KUKA KRL program: EPS_2_25694_LG04A_A_20260223033044.src

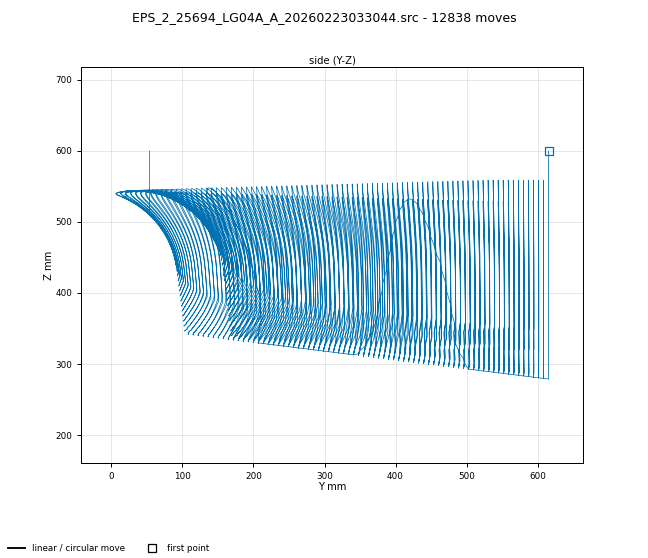
[picture p0: tool path of EPS_2_25694_LG04A_A_20260223033044.src, 12838 of 12840 moves have a stored position in this frame; points joined in program order, loops and branches not executed]
&ACCESS RVP
&REL 4
&COMMENT QRS 19112012
&PARAM EDITMASK = *
DEF PART()
EXT BAS (BAS_COMMAND :IN,REAL :IN )
INT I
BAS (#INITMOV,0 )

;KUKA QRS Post kuka4.cps  Date:22-06-2017 !

File_ID=3043

QRS_PRE_INIT()

;Init var - Until changes are made in qrs_pre_init
Outlet_Square_prg=0
Inlet_1_Square_prg=0
Inlet_2_Square_prg=0
Inlet_3_Square_prg=0
Inlet_4_Square_prg=0
Inlet_5_Square_prg=0

Outlet_1={X 0.000, Y 535.490, Z 458.500, B 0.000, E1 0.000 }
Inlet_1={X 0.000, Y 537.630, Z 428.500, B 0.000, E1 169.000 }
Outlet_1_type=201
Inlet_1_type=201
;QRS#1=Sidecore dimensions
;QRS#2=200-8" PVC SDR 35
;QRS#3=200-8" PVC SDR 35
;QRS#4=
;QRS#5=
;QRS#6=
;QRS#7=
;QRS#8=
;QRS#9=12-08 PSX
;QRS#10=12-08 PSX
;QRS#11=
;QRS#12=
;QRS#13=
;QRS#14=
;QRS#15=
;QRS#16=1220x127x838 2,75'
;QRS#17=EPS Height
;QRS#18=559
;QRS#19=*
;QRS#20= UPDATED VERSION 22-06-2017
;QRS#21=*
Outlet_Square=0100
Inlet_1_Square=0100
Inlet_2_Square=0
Inlet_3_Square=0
Inlet_4_Square=0
Inlet_5_Square=0
Mill_Square=1
Outlet_Square_Prg=204
Inlet_1_Square_prg=204

QRS_INIT()

$ADVANCE=5

; T1
PTP {E1 173.619,E2 173.619}
PTP {X 0,Y 615.493,A -85,B 0,C 180,E1 173.619,E2 173.619,E3 0,E4 0,E5 0,E6 0}
QRS_SPEED_INIT()
LIN {X 0,Y 615.493,Z 600,A -85,B 0,C 180,E1 173.619,E2 173.619,E3 0,E4 0,E5 0,E6 0} C_VEL
LIN {X 0,Y 615.493,Z 288.877,A -85,B 0,C 180,E1 173.619,E2 173.619} C_VEL
LIN {X 0,Y 615.493,Z 280.697,A -85,B 0,C 180,E1 173.619,E2 173.619} C_VEL
LIN {X 0,Y 615.473,Z 278.697,A -85,B 0,C 180,E1 173.433,E2 173.433} C_VEL
LIN {X 0,Y 615.45,Z 278.69,A -85,B 0,C 180,E1 170.8,E2 170.8} C_VEL
LIN {X 0,Y 615.482,Z 278.684,A -85,B 0,C 180,E1 168.139,E2 168.139} C_VEL
LIN {X 0,Y 615.489,Z 278.699,A -85,B 0,C 180,E1 165.451,E2 165.451} C_VEL
LIN {X 0,Y 615.451,Z 278.694,A -85,B 0,C 180,E1 162.728,E2 162.728} C_VEL
LIN {X 0,Y 615.453,Z 278.693,A -85,B 0,C 180,E1 160.661,E2 160.661} C_VEL
LIN {X 0,Y 615.452,Z 278.693,A -85,B 0,C 180,E1 158.567,E2 158.567} C_VEL
LIN {X 0,Y 615.457,Z 278.687,A -85,B 0,C 180,E1 155.998,E2 155.998} C_VEL
LIN {X 0,Y 615.483,Z 278.684,A -85,B 0,C 180,E1 153.555,E2 153.555} C_VEL
LIN {X 0,Y 615.473,Z 278.698,A -85,B 0,C 180,E1 150.593,E2 150.593} C_VEL
LIN {X 0,Y 615.456,Z 278.696,A -85,B 0,C 180,E1 148.312,E2 148.312} C_VEL
LIN {X 0,Y 615.447,Z 278.692,A -85,B 0,C 180,E1 145.975,E2 145.975} C_VEL
LIN {X 0,Y 615.453,Z 278.688,A -85,B 0,C 180,E1 143.572,E2 143.572} C_VEL
LIN {X 0,Y 615.494,Z 278.684,A -85,B 0,C 180,E1 140.937,E2 140.937} C_VEL
LIN {X 0,Y 615.49,Z 278.695,A -85,B 0,C 180,E1 138.526,E2 138.526} C_VEL
LIN {X 0,Y 615.459,Z 278.695,A -85,B 0,C 180,E1 135.847,E2 135.847} C_VEL
LIN {X 0,Y 615.448,Z 278.689,A -85,B 0,C 180,E1 133.248,E2 133.248} C_VEL
LIN {X 0,Y 615.488,Z 278.684,A -85,B 0,C 180,E1 130.607,E2 130.607} C_VEL
LIN {X 0,Y 615.485,Z 278.7,A -85,B 0,C 180,E1 128.011,E2 128.011} C_VEL
LIN {X 0,Y 615.472,Z 278.697,A -85,B 0,C 180,E1 125.617,E2 125.617} C_VEL
LIN {X 0,Y 615.451,Z 278.694,A -85,B 0,C 180,E1 123.239,E2 123.239} C_VEL
LIN {X 0,Y 615.458,Z 278.687,A -85,B 0,C 180,E1 120.541,E2 120.541} C_VEL
LIN {X 0,Y 615.492,Z 278.741,A -85,B 0,C 180,E1 120.207,E2 120.207} C_VEL
LIN {X 0,Y 615.495,Z 297.187,A -85,B 0,C 180,E1 117.177,E2 117.177} C_VEL
LIN {X 0,Y 615.475,Z 314.006,A -85,B 0,C 180,E1 114.452,E2 114.452} C_VEL
LIN {X 0,Y 615.494,Z 318.036,A -85,B 0,C 180,E1 113.809,E2 113.809} C_VEL
LIN {X 0,Y 615.476,Z 425.627,A -85,B 0,C 180,E1 112.53,E2 112.53} C_VEL
LIN {X 0,Y 615.474,Z 438.589,A -85,B 0,C 180,E1 112.239,E2 112.239} C_VEL
LIN {X 0,Y 615.497,Z 450.996,A -85,B 0,C 180,E1 111.828,E2 111.828} C_VEL
LIN {X 0,Y 615.482,Z 463.588,A -85,B 0,C 180,E1 111.257,E2 111.257} C_VEL
LIN {X 0,Y 615.496,Z 475.428,A -85,B 0,C 180,E1 110.558,E2 110.558} C_VEL
LIN {X 0,Y 615.498,Z 483.736,A -85,B 0,C 180,E1 109.946,E2 109.946} C_VEL
LIN {X 0,Y 615.498,Z 490.882,A -85,B 0,C 180,E1 109.338,E2 109.338} C_VEL
LIN {X 0,Y 615.496,Z 499.643,A -85,B 0,C 180,E1 108.444,E2 108.444} C_VEL
LIN {X 0,Y 615.493,Z 507.562,A -85,B 0,C 180,E1 107.442,E2 107.442} C_VEL
LIN {X 0,Y 615.496,Z 513.912,A -85,B 0,C 180,E1 106.432,E2 106.432} C_VEL
LIN {X 0,Y 615.497,Z 519.787,A -85,B 0,C 180,E1 105.226,E2 105.226} C_VEL
LIN {X 0,Y 615.496,Z 522.37,A -85,B 0,C 180,E1 104.549,E2 104.549} C_VEL
LIN {X 0,Y 615.496,Z 524.427,A -85,B 0,C 180,E1 103.874,E2 103.874} C_VEL
LIN {X 0,Y 615.495,Z 526.05,A -85,B 0,C 180,E1 103.201,E2 103.201} C_VEL
LIN {X 0,Y 615.497,Z 527.253,A -85,B 0,C 180,E1 102.53,E2 102.53} C_VEL
LIN {X 0,Y 615.494,Z 527.997,A -85,B 0,C 180,E1 101.861,E2 101.861} C_VEL
LIN {X 0,Y 615.497,Z 528.293,A -85,B 0,C 180,E1 100.527,E2 100.527} C_VEL
LIN {X 0,Y 615.496,Z 527.836,A -85,B 0,C 180,E1 99.862,E2 99.862} C_VEL
LIN {X 0,Y 615.495,Z 525.678,A -85,B 0,C 180,E1 98.537,E2 98.537} C_VEL
LIN {X 0,Y 615.495,Z 522.962,A -85,B 0,C 180,E1 97.546,E2 97.546} C_VEL
LIN {X 0,Y 615.497,Z 519.242,A -85,B 0,C 180,E1 96.557,E2 96.557} C_VEL
LIN {X 0,Y 615.497,Z 514.417,A -85,B 0,C 180,E1 95.57,E2 95.57} C_VEL
LIN {X 0,Y 615.495,Z 508.351,A -85,B 0,C 180,E1 94.585,E2 94.585} C_VEL
LIN {X 0,Y 615.493,Z 500.832,A -85,B 0,C 180,E1 93.601,E2 93.601} C_VEL
LIN {X 0,Y 615.498,Z 493.027,A -85,B 0,C 180,E1 92.782,E2 92.782} C_VEL
LIN {X 0,Y 615.497,Z 485.721,A -85,B 0,C 180,E1 92.127,E2 92.127} C_VEL
LIN {X 0,Y 615.486,Z 477.224,A -85,B 0,C 180,E1 91.473,E2 91.473} C_VEL
LIN {X 0,Y 615.483,Z 466.689,A -85,B 0,C 180,E1 90.818,E2 90.818} C_VEL
LIN {X 0,Y 615.492,Z 454.96,A -85,B 0,C 180,E1 90.246,E2 90.246} C_VEL
LIN {X 0,Y 615.484,Z 442.825,A -85,B 0,C 180,E1 89.796,E2 89.796} C_VEL
LIN {X 0,Y 615.474,Z 430.38,A -85,B 0,C 180,E1 89.469,E2 89.469} C_VEL
LIN {X 0,Y 615.478,Z 415.696,A -85,B 0,C 180,E1 89.244,E2 89.244} C_VEL
LIN {X 0,Y 615.496,Z 317.979,A -85,B 0,C 180,E1 88.099,E2 88.099} C_VEL
LIN {X 0,Y 615.475,Z 300.382,A -85,B 0,C 180,E1 85.252,E2 85.252} C_VEL
LIN {X 0,Y 615.496,Z 283.292,A -85,B 0,C 180,E1 82.455,E2 82.455} C_VEL
LIN {X 0,Y 615.44,Z 278.695,A -85,B 0,C 180,E1 81.67,E2 81.67} C_VEL
LIN {X 0,Y 615.441,Z 278.691,A -85,B 0,C 180,E1 79.137,E2 79.137} C_VEL
LIN {X 0,Y 615.457,Z 278.69,A -85,B 0,C 180,E1 76.799,E2 76.799} C_VEL
LIN {X 0,Y 615.491,Z 278.699,A -85,B 0,C 180,E1 74.096,E2 74.096} C_VEL
LIN {X 0,Y 615.436,Z 278.696,A -85,B 0,C 180,E1 71.353,E2 71.353} C_VEL
LIN {X 0,Y 615.435,Z 278.696,A -85,B 0,C 180,E1 69.268,E2 69.268} C_VEL
LIN {X 0,Y 615.432,Z 278.696,A -85,B 0,C 180,E1 67.154,E2 67.154} C_VEL
LIN {X 0,Y 615.428,Z 278.695,A -85,B 0,C 180,E1 65.006,E2 65.006} C_VEL
LIN {X 0,Y 615.425,Z 278.695,A -85,B 0,C 180,E1 62.821,E2 62.821} C_VEL
LIN {X 0,Y 615.426,Z 278.694,A -85,B 0,C 180,E1 60.591,E2 60.591} C_VEL
LIN {X 0,Y 615.431,Z 278.694,A -85,B 0,C 180,E1 58.312,E2 58.312} C_VEL
LIN {X 0,Y 615.456,Z 278.693,A -85,B 0,C 180,E1 55.977,E2 55.977} C_VEL
LIN {X 0,Y 615.456,Z 278.699,A -85,B 0,C 180,E1 53.068,E2 53.068} C_VEL
LIN {X 0,Y 615.419,Z 278.696,A -85,B 0,C 180,E1 50.246,E2 50.246} C_VEL
LIN {X 0,Y 615.455,Z 278.694,A -85,B 0,C 180,E1 47.645,E2 47.645} C_VEL
LIN {X 0,Y 615.472,Z 278.7,A -85,B 0,C 180,E1 44.931,E2 44.931} C_VEL
LIN {X 0,Y 615.42,Z 278.698,A -85,B 0,C 180,E1 42.359,E2 42.359} C_VEL
LIN {X 0,Y 615.41,Z 278.698,A -85,B 0,C 180,E1 40.082,E2 40.082} C_VEL
LIN {X 0,Y 615.41,Z 278.698,A -85,B 0,C 180,E1 38.004,E2 38.004} C_VEL
LIN {X 0,Y 615.413,Z 278.698,A -85,B 0,C 180,E1 35.621,E2 35.621} C_VEL
LIN {X 0,Y 615.434,Z 278.698,A -85,B 0,C 180,E1 33.24,E2 33.24} C_VEL
LIN {X 0,Y 615.431,Z 278.7,A -85,B 0,C 180,E1 30.164,E2 30.164} C_VEL
LIN {X 0,Y 615.415,Z 278.7,A -85,B 0,C 180,E1 27.919,E2 27.919} C_VEL
LIN {X 0,Y 615.402,Z 278.7,A -85,B 0,C 180,E1 25.554,E2 25.554} C_VEL
LIN {X 0,Y 615.403,Z 278.7,A -85,B 0,C 180,E1 23.56,E2 23.56} C_VEL
LIN {X 0,Y 615.403,Z 278.7,A -85,B 0,C 180,E1 21.435,E2 21.435} C_VEL
LIN {X 0,Y 615.403,Z 278.7,A -85,B 0,C 180,E1 19.341,E2 19.341} C_VEL
LIN {X 0,Y 615.405,Z 278.699,A -85,B 0,C 180,E1 17.273,E2 17.273} C_VEL
LIN {X 0,Y 615.407,Z 278.699,A -85,B 0,C 180,E1 15.228,E2 15.228} C_VEL
LIN {X 0,Y 615.41,Z 278.698,A -85,B 0,C 180,E1 13.203,E2 13.203} C_VEL
LIN {X 0,Y 615.41,Z 278.698,A -85,B 0,C 180,E1 10.856,E2 10.856} C_VEL
LIN {X 0,Y 615.423,Z 278.699,A -85,B 0,C 180,E1 8.538,E2 8.538} C_VEL
LIN {X 0,Y 615.493,Z 278.7,A -85,B 0,C 180,E1 5.899,E2 5.899} C_VEL
LIN {X 0,Y 615.447,Z 278.695,A -85,B 0,C 180,E1 3.273,E2 3.273} C_VEL
LIN {X 0,Y 615.416,Z 278.697,A -85,B 0,C 180,E1 0.654,E2 0.654} C_VEL
LIN {X 0,Y 615.419,Z 278.696,A -85,B 0,C 180,E1 -1.309,E2 -1.309} C_VEL
LIN {X 0,Y 615.425,Z 278.695,A -85,B 0,C 180,E1 -3.273,E2 -3.273} C_VEL
LIN {X 0,Y 615.431,Z 278.695,A -85,B 0,C 180,E1 -5.242,E2 -5.242} C_VEL
LIN {X 0,Y 615.441,Z 278.694,A -85,B 0,C 180,E1 -7.216,E2 -7.216} C_VEL
LIN {X 0,Y 615.452,Z 278.693,A -85,B 0,C 180,E1 -9.199,E2 -9.199} C_VEL
LIN {X 0,Y 615.462,Z 278.692,A -85,B 0,C 180,E1 -11.193,E2 -11.193} C_VEL
LIN {X 0,Y 615.425,Z 278.695,A -85,B 0,C 180,E1 -13.913,E2 -13.913} C_VEL
LIN {X 0,Y 615.444,Z 278.697,A -85,B 0,C 180,E1 -16.421,E2 -16.421} C_VEL
LIN {X 0,Y 615.482,Z 278.69,A -85,B 0,C 180,E1 -19.338,E2 -19.338} C_VEL
LIN {X 0,Y 615.43,Z 278.694,A -85,B 0,C 180,E1 -22.139,E2 -22.139} C_VEL
LIN {X 0,Y 615.43,Z 278.694,A -85,B 0,C 180,E1 -24.274,E2 -24.274} C_VEL
LIN {X 0,Y 615.433,Z 278.694,A -85,B 0,C 180,E1 -26.447,E2 -26.447} C_VEL
LIN {X 0,Y 615.492,Z 278.696,A -85,B 0,C 180,E1 -29.406,E2 -29.406} C_VEL
LIN {X 0,Y 615.441,Z 278.691,A -85,B 0,C 180,E1 -32.326,E2 -32.326} C_VEL
LIN {X 0,Y 615.437,Z 278.693,A -85,B 0,C 180,E1 -34.696,E2 -34.696} C_VEL
LIN {X 0,Y 615.464,Z 278.697,A -85,B 0,C 180,E1 -37.244,E2 -37.244} C_VEL
LIN {X 0,Y 615.495,Z 278.685,A -85,B 0,C 180,E1 -40.091,E2 -40.091} C_VEL
LIN {X 0,Y 615.469,Z 278.687,A -85,B 0,C 180,E1 -42.355,E2 -42.355} C_VEL
LIN {X 0,Y 615.442,Z 278.691,A -85,B 0,C 180,E1 -44.928,E2 -44.928} C_VEL
LIN {X 0,Y 615.443,Z 278.691,A -85,B 0,C 180,E1 -46.957,E2 -46.957} C_VEL
LIN {X 0,Y 615.448,Z 278.695,A -85,B 0,C 180,E1 -49.392,E2 -49.392} C_VEL
LIN {X 0,Y 615.482,Z 278.704,A -85,B 0,C 180,E1 -51.989,E2 -51.989} C_VEL
LIN {X 0,Y 615.493,Z 278.69,A -85,B 0,C 180,E1 -54.386,E2 -54.386} C_VEL
LIN {X 0,Y 615.485,Z 278.684,A -85,B 0,C 180,E1 -56.765,E2 -56.765} C_VEL
LIN {X 0,Y 615.468,Z 278.685,A -85,B 0,C 180,E1 -59.08,E2 -59.08} C_VEL
LIN {X 0,Y 615.451,Z 278.69,A -85,B 0,C 180,E1 -61.556,E2 -61.556} C_VEL
LIN {X 0,Y 615.451,Z 278.689,A -85,B 0,C 180,E1 -63.555,E2 -63.555} C_VEL
LIN {X 0,Y 615.459,Z 278.694,A -85,B 0,C 180,E1 -65.998,E2 -65.998} C_VEL
LIN {X 0,Y 615.454,Z 278.771,A -85,B 0,C 180,E1 -67.838,E2 -67.838} C_VEL
LIN {X 0,Y 615.483,Z 297.824,A -85,B 0,C 180,E1 -70.489,E2 -70.489} C_VEL
LIN {X 0,Y 615.496,Z 319.189,A -85,B 0,C 180,E1 -73.414,E2 -73.414} C_VEL
LIN {X 0,Y 615.486,Z 340.532,A -85,B 0,C 180,E1 -76.295,E2 -76.295} C_VEL
LIN {X 0,Y 615.476,Z 346.647,A -85,B 0,C 180,E1 -77.114,E2 -77.114} C_VEL
LIN {X 0,Y 615.488,Z 454.864,A -85,B 0,C 180,E1 -78.411,E2 -78.411} C_VEL
LIN {X 0,Y 615.493,Z 467.365,A -85,B 0,C 180,E1 -78.683,E2 -78.683} C_VEL
LIN {X 0,Y 615.492,Z 480.561,A -85,B 0,C 180,E1 -79.111,E2 -79.111} C_VEL
LIN {X 0,Y 615.489,Z 492.488,A -85,B 0,C 180,E1 -79.64,E2 -79.64} C_VEL
LIN {X 0,Y 615.478,Z 504.006,A -85,B 0,C 180,E1 -80.304,E2 -80.304} C_VEL
LIN {X 0,Y 615.498,Z 513.228,A -85,B 0,C 180,E1 -80.968,E2 -80.968} C_VEL
LIN {X 0,Y 615.498,Z 521.008,A -85,B 0,C 180,E1 -81.629,E2 -81.629} C_VEL
LIN {X 0,Y 615.497,Z 530.611,A -85,B 0,C 180,E1 -82.62,E2 -82.62} C_VEL
LIN {X 0,Y 615.49,Z 538.208,A -85,B 0,C 180,E1 -83.609,E2 -83.609} C_VEL
LIN {X 0,Y 615.498,Z 545.207,A -85,B 0,C 180,E1 -84.759,E2 -84.759} C_VEL
LIN {X 0,Y 615.493,Z 549.854,A -85,B 0,C 180,E1 -85.744,E2 -85.744} C_VEL
LIN {X 0,Y 615.496,Z 553.4,A -85,B 0,C 180,E1 -86.728,E2 -86.728} C_VEL
LIN {X 0,Y 615.497,Z 555.234,A -85,B 0,C 180,E1 -87.383,E2 -87.383} C_VEL
LIN {X 0,Y 615.496,Z 556.609,A -85,B 0,C 180,E1 -88.037,E2 -88.037} C_VEL
LIN {X 0,Y 615.496,Z 558.174,A -85,B 0,C 180,E1 -89.346,E2 -89.346} C_VEL
LIN {X 0,Y 615.494,Z 558.389,A -85,B 0,C 180,E1 -90,E2 -90} C_VEL
LIN {X 0,Y 615.496,Z 557.579,A -85,B 0,C 180,E1 -91.309,E2 -91.309} C_VEL
LIN {X 0,Y 615.496,Z 556.607,A -85,B 0,C 180,E1 -91.964,E2 -91.964} C_VEL
LIN {X 0,Y 615.497,Z 555.232,A -85,B 0,C 180,E1 -92.618,E2 -92.618} C_VEL
LIN {X 0,Y 615.496,Z 552.348,A -85,B 0,C 180,E1 -93.601,E2 -93.601} C_VEL
LIN {X 0,Y 615.498,Z 548.44,A -85,B 0,C 180,E1 -94.585,E2 -94.585} C_VEL
LIN {X 0,Y 615.499,Z 543.402,A -85,B 0,C 180,E1 -95.57,E2 -95.57} C_VEL
LIN {X 0,Y 615.489,Z 536.916,A -85,B 0,C 180,E1 -96.577,E2 -96.577} C_VEL
LIN {X 0,Y 615.497,Z 529.129,A -85,B 0,C 180,E1 -97.546,E2 -97.546} C_VEL
LIN {X 0,Y 615.498,Z 519.253,A -85,B 0,C 180,E1 -98.537,E2 -98.537} C_VEL
LIN {X 0,Y 615.492,Z 507.705,A -85,B 0,C 180,E1 -99.448,E2 -99.448} C_VEL
LIN {X 0,Y 615.48,Z 497.148,A -85,B 0,C 180,E1 -100.112,E2 -100.112} C_VEL
LIN {X 0,Y 615.496,Z 484.986,A -85,B 0,C 180,E1 -100.708,E2 -100.708} C_VEL
LIN {X 0,Y 615.489,Z 472.933,A -85,B 0,C 180,E1 -101.155,E2 -101.155} C_VEL
LIN {X 0,Y 615.491,Z 460.398,A -85,B 0,C 180,E1 -101.485,E2 -101.485} C_VEL
LIN {X 0,Y 615.487,Z 447.127,A -85,B 0,C 180,E1 -101.694,E2 -101.694} C_VEL
LIN {X 0,Y 615.475,Z 346.64,A -85,B 0,C 180,E1 -102.887,E2 -102.887} C_VEL
LIN {X 0,Y 615.496,Z 325.462,A -85,B 0,C 180,E1 -105.735,E2 -105.735} C_VEL
LIN {X 0,Y 615.486,Z 304.105,A -85,B 0,C 180,E1 -108.646,E2 -108.646} C_VEL
LIN {X 0,Y 615.497,Z 283.978,A -85,B 0,C 180,E1 -111.432,E2 -111.432} C_VEL
LIN {X 0,Y 615.454,Z 278.69,A -85,B 0,C 180,E1 -112.188,E2 -112.188} C_VEL
LIN {X 0,Y 615.492,Z 278.682,A -85,B 0,C 180,E1 -114.992,E2 -114.992} C_VEL
LIN {X 0,Y 615.478,Z 278.697,A -85,B 0,C 180,E1 -117.916,E2 -117.916} C_VEL
LIN {X 0,Y 615.465,Z 278.695,A -85,B 0,C 180,E1 -120.162,E2 -120.162} C_VEL
LIN {X 0,Y 615.455,Z 278.692,A -85,B 0,C 180,E1 -122.46,E2 -122.46} C_VEL
LIN {X 0,Y 615.455,Z 278.688,A -85,B 0,C 180,E1 -124.817,E2 -124.817} C_VEL
LIN {X 0,Y 615.476,Z 278.683,A -85,B 0,C 180,E1 -127.243,E2 -127.243} C_VEL
LIN {X 0,Y 615.495,Z 278.697,A -85,B 0,C 180,E1 -130.09,E2 -130.09} C_VEL
LIN {X 0,Y 615.49,Z 278.699,A -85,B 0,C 180,E1 -132.353,E2 -132.353} C_VEL
LIN {X 0,Y 615.45,Z 278.691,A -85,B 0,C 180,E1 -135.072,E2 -135.072} C_VEL
LIN {X 0,Y 615.497,Z 278.682,A -85,B 0,C 180,E1 -137.919,E2 -137.919} C_VEL
LIN {X 0,Y 615.49,Z 278.69,A -85,B 0,C 180,E1 -140.25,E2 -140.25} C_VEL
LIN {X 0,Y 615.462,Z 278.695,A -85,B 0,C 180,E1 -143.067,E2 -143.067} C_VEL
LIN {X 0,Y 615.454,Z 278.693,A -85,B 0,C 180,E1 -145.304,E2 -145.304} C_VEL
LIN {X 0,Y 615.453,Z 278.689,A -85,B 0,C 180,E1 -147.674,E2 -147.674} C_VEL
LIN {X 0,Y 615.482,Z 278.683,A -85,B 0,C 180,E1 -150.206,E2 -150.206} C_VEL
LIN {X 0,Y 615.492,Z 278.697,A -85,B 0,C 180,E1 -152.954,E2 -152.954} C_VEL
LIN {X 0,Y 615.452,Z 278.692,A -85,B 0,C 180,E1 -155.726,E2 -155.726} C_VEL
LIN {X 0,Y 615.452,Z 278.692,A -85,B 0,C 180,E1 -157.862,E2 -157.862} C_VEL
LIN {X 0,Y 615.45,Z 278.692,A -85,B 0,C 180,E1 -159.966,E2 -159.966} C_VEL
LIN {X 0,Y 615.451,Z 278.691,A -85,B 0,C 180,E1 -162.042,E2 -162.042} C_VEL
LIN {X 0,Y 615.483,Z 278.683,A -85,B 0,C 180,E1 -164.774,E2 -164.774} C_VEL
LIN {X 0,Y 615.489,Z 278.697,A -85,B 0,C 180,E1 -167.47,E2 -167.47} C_VEL
LIN {X 0,Y 615.458,Z 278.694,A -85,B 0,C 180,E1 -170.137,E2 -170.137} C_VEL
LIN {X 0,Y 615.458,Z 278.687,A -85,B 0,C 180,E1 -172.784,E2 -172.784} C_VEL
LIN {X 0,Y 615.495,Z 278.684,A -85,B 0,C 180,E1 -175.416,E2 -175.416} C_VEL
LIN {X 0,Y 615.496,Z 278.7,A -85,B 0,C 180,E1 -178.037,E2 -178.037} C_VEL
LIN {X 0,Y 615.453,Z 278.693,A -85,B 0,C 180,E1 -180.654,E2 -180.654} C_VEL
LIN {X 0,Y 615.462,Z 278.686,A -85,B 0,C 180,E1 -183.273,E2 -183.273} C_VEL
LIN {X 0,Y 615.493,Z 278.687,A -85,B 0,C 180,E1 -185.899,E2 -185.899} C_VEL
LIN {X 0,Y 615.473,Z 278.697,A -85,B 0,C 180,E1 -186.567,E2 -186.567} C_VEL
LIN {X 0,Y 614.78,Z 278.837,A -85,B 0,C 180,E1 -187.113,E2 -187.113} C_VEL
LIN {X 0,Y 611.93,Z 279.257,A -85,B 0,C 180,E1 -187.999,E2 -187.999} C_VEL
LIN {X 0,Y 609.542,Z 279.564,A -85,B 0,C 180,E1 -188.712,E2 -188.712} C_VEL
LIN {X 0,Y 608.522,Z 279.679,A -85,B 0,C 180,E1 -189.261,E2 -189.261} C_VEL
LIN {X 0,Y 608.441,Z 279.687,A -85,B 0,C 180,E1 -189.447,E2 -189.447} C_VEL
LIN {X 0,Y 608.46,Z 279.688,A -85,B 0,C 180,E1 -192,E2 -192} C_VEL
LIN {X 0,Y 608.469,Z 279.695,A -85,B 0,C 180,E1 -194.721,E2 -194.721} C_VEL
LIN {X 0,Y 608.425,Z 279.69,A -85,B 0,C 180,E1 -197.478,E2 -197.478} C_VEL
LIN {X 0,Y 608.428,Z 279.69,A -85,B 0,C 180,E1 -199.572,E2 -199.572} C_VEL
LIN {X 0,Y 608.443,Z 279.688,A -85,B 0,C 180,E1 -201.693,E2 -201.693} C_VEL
LIN {X 0,Y 608.454,Z 279.69,A -85,B 0,C 180,E1 -204.571,E2 -204.571} C_VEL
LIN {X 0,Y 608.435,Z 279.693,A -85,B 0,C 180,E1 -207.519,E2 -207.519} C_VEL
LIN {X 0,Y 608.419,Z 279.691,A -85,B 0,C 180,E1 -209.964,E2 -209.964} C_VEL
LIN {X 0,Y 608.445,Z 279.687,A -85,B 0,C 180,E1 -212.52,E2 -212.52} C_VEL
LIN {X 0,Y 608.442,Z 279.696,A -85,B 0,C 180,E1 -215.278,E2 -215.278} C_VEL
LIN {X 0,Y 608.452,Z 279.694,A -85,B 0,C 180,E1 -217.748,E2 -217.748} C_VEL
LIN {X 0,Y 608.435,Z 279.689,A -85,B 0,C 180,E1 -220.327,E2 -220.327} C_VEL
LIN {X 0,Y 608.483,Z 279.686,A -85,B 0,C 180,E1 -223.31,E2 -223.31} C_VEL
LIN {X 0,Y 608.459,Z 279.692,A -85,B 0,C 180,E1 -226.129,E2 -226.129} C_VEL
LIN {X 0,Y 608.421,Z 279.69,A -85,B 0,C 180,E1 -228.82,E2 -228.82} C_VEL
LIN {X 0,Y 608.465,Z 279.691,A -85,B 0,C 180,E1 -231.761,E2 -231.761} C_VEL
LIN {X 0,Y 608.425,Z 279.692,A -85,B 0,C 180,E1 -234.721,E2 -234.721} C_VEL
LIN {X 0,Y 608.453,Z 279.687,A -85,B 0,C 180,E1 -237.48,E2 -237.48} C_VEL
LIN {X 0,Y 608.492,Z 279.837,A -85,B 0,C 180,E1 -239.737,E2 -239.737} C_VEL
LIN {X 0,Y 608.484,Z 296.397,A -85,B 0,C 180,E1 -242.483,E2 -242.483} C_VEL
LIN {X 0,Y 608.46,Z 313.301,A -85,B 0,C 180,E1 -245.247,E2 -245.247} C_VEL
LIN {X 0,Y 608.462,Z 318.194,A -85,B 0,C 180,E1 -246.041,E2 -246.041} C_VEL
LIN {X 0,Y 608.525,Z 425.131,A -85,B 0,C 180,E1 -247.325,E2 -247.325} C_VEL
LIN {X 0,Y 608.516,Z 438.538,A -85,B 0,C 180,E1 -247.626,E2 -247.626} C_VEL
LIN {X 0,Y 608.534,Z 451.048,A -85,B 0,C 180,E1 -248.043,E2 -248.043} C_VEL
LIN {X 0,Y 608.488,Z 462.858,A -85,B 0,C 180,E1 -248.576,E2 -248.576} C_VEL
LIN {X 0,Y 608.512,Z 473.869,A -85,B 0,C 180,E1 -249.215,E2 -249.215} C_VEL
LIN {X 0,Y 608.477,Z 483.424,A -85,B 0,C 180,E1 -249.902,E2 -249.902} C_VEL
LIN {X 0,Y 608.487,Z 491.598,A -85,B 0,C 180,E1 -250.606,E2 -250.606} C_VEL
LIN {X 0,Y 608.474,Z 500.264,A -85,B 0,C 180,E1 -251.5,E2 -251.5} C_VEL
LIN {X 0,Y 608.448,Z 508.244,A -85,B 0,C 180,E1 -252.523,E2 -252.523} C_VEL
LIN {X 0,Y 608.434,Z 514.264,A -85,B 0,C 180,E1 -253.483,E2 -253.483} C_VEL
LIN {X 0,Y 608.427,Z 519.744,A -85,B 0,C 180,E1 -254.593,E2 -254.593} C_VEL
LIN {X 0,Y 608.428,Z 523.592,A -85,B 0,C 180,E1 -255.62,E2 -255.62} C_VEL
LIN {X 0,Y 608.438,Z 526.355,A -85,B 0,C 180,E1 -256.643,E2 -256.643} C_VEL
LIN {X 0,Y 608.42,Z 527.637,A -85,B 0,C 180,E1 -257.322,E2 -257.322} C_VEL
LIN {X 0,Y 608.44,Z 528.506,A -85,B 0,C 180,E1 -257.999,E2 -257.999} C_VEL
LIN {X 0,Y 608.448,Z 529,A -85,B 0,C 180,E1 -259.057,E2 -259.057} C_VEL
LIN {X 0,Y 608.432,Z 528.562,A -85,B 0,C 180,E1 -260.022,E2 -260.022} C_VEL
LIN {X 0,Y 608.423,Z 527.762,A -85,B 0,C 180,E1 -260.693,E2 -260.693} C_VEL
LIN {X 0,Y 608.421,Z 526.538,A -85,B 0,C 180,E1 -261.363,E2 -261.363} C_VEL
LIN {X 0,Y 608.424,Z 523.924,A -85,B 0,C 180,E1 -262.366,E2 -262.366} C_VEL
LIN {X 0,Y 608.453,Z 519.172,A -85,B 0,C 180,E1 -263.631,E2 -263.631} C_VEL
LIN {X 0,Y 608.462,Z 513.763,A -85,B 0,C 180,E1 -264.698,E2 -264.698} C_VEL
LIN {X 0,Y 608.438,Z 507.355,A -85,B 0,C 180,E1 -265.694,E2 -265.694} C_VEL
LIN {X 0,Y 608.451,Z 499.384,A -85,B 0,C 180,E1 -266.689,E2 -266.689} C_VEL
LIN {X 0,Y 608.484,Z 489.512,A -85,B 0,C 180,E1 -267.683,E2 -267.683} C_VEL
LIN {X 0,Y 608.471,Z 478.058,A -85,B 0,C 180,E1 -268.593,E2 -268.593} C_VEL
LIN {X 0,Y 608.498,Z 467.652,A -85,B 0,C 180,E1 -269.255,E2 -269.255} C_VEL
LIN {X 0,Y 608.509,Z 456.141,A -85,B 0,C 180,E1 -269.834,E2 -269.834} C_VEL
LIN {X 0,Y 608.517,Z 443.034,A -85,B 0,C 180,E1 -270.33,E2 -270.33} C_VEL
LIN {X 0,Y 608.516,Z 430.618,A -85,B 0,C 180,E1 -270.661,E2 -270.661} C_VEL
LIN {X 0,Y 608.53,Z 417.842,A -85,B 0,C 180,E1 -270.868,E2 -270.868} C_VEL
LIN {X 0,Y 608.498,Z 318.287,A -85,B 0,C 180,E1 -272.047,E2 -272.047} C_VEL
LIN {X 0,Y 608.471,Z 301.29,A -85,B 0,C 180,E1 -274.803,E2 -274.803} C_VEL
LIN {X 0,Y 608.514,Z 284.155,A -85,B 0,C 180,E1 -277.632,E2 -277.632} C_VEL
LIN {X 0,Y 608.42,Z 279.693,A -85,B 0,C 180,E1 -278.385,E2 -278.385} C_VEL
LIN {X 0,Y 608.437,Z 279.688,A -85,B 0,C 180,E1 -280.938,E2 -280.938} C_VEL
LIN {X 0,Y 608.48,Z 279.692,A -85,B 0,C 180,E1 -284.019,E2 -284.019} C_VEL
LIN {X 0,Y 608.414,Z 279.692,A -85,B 0,C 180,E1 -286.784,E2 -286.784} C_VEL
LIN {X 0,Y 608.433,Z 279.691,A -85,B 0,C 180,E1 -289.57,E2 -289.57} C_VEL
LIN {X 0,Y 608.431,Z 279.695,A -85,B 0,C 180,E1 -292.469,E2 -292.469} C_VEL
LIN {X 0,Y 608.432,Z 279.694,A -85,B 0,C 180,E1 -294.571,E2 -294.571} C_VEL
LIN {X 0,Y 608.41,Z 279.692,A -85,B 0,C 180,E1 -297.194,E2 -297.194} C_VEL
LIN {X 0,Y 608.449,Z 279.69,A -85,B 0,C 180,E1 -299.968,E2 -299.968} C_VEL
LIN {X 0,Y 608.431,Z 279.694,A -85,B 0,C 180,E1 -302.88,E2 -302.88} C_VEL
LIN {X 0,Y 608.401,Z 279.694,A -85,B 0,C 180,E1 -305.279,E2 -305.279} C_VEL
LIN {X 0,Y 608.402,Z 279.693,A -85,B 0,C 180,E1 -307.75,E2 -307.75} C_VEL
LIN {X 0,Y 608.43,Z 279.693,A -85,B 0,C 180,E1 -310.326,E2 -310.326} C_VEL
LIN {X 0,Y 608.434,Z 279.692,A -85,B 0,C 180,E1 -313.305,E2 -313.305} C_VEL
LIN {X 0,Y 608.396,Z 279.694,A -85,B 0,C 180,E1 -315.741,E2 -315.741} C_VEL
LIN {X 0,Y 608.397,Z 279.693,A -85,B 0,C 180,E1 -317.933,E2 -317.933} C_VEL
LIN {X 0,Y 608.428,Z 279.694,A -85,B 0,C 180,E1 -320.706,E2 -320.706} C_VEL
LIN {X 0,Y 608.445,Z 279.698,A -85,B 0,C 180,E1 -323.084,E2 -323.084} C_VEL
LIN {X 0,Y 608.447,Z 279.693,A -85,B 0,C 180,E1 -325.529,E2 -325.529} C_VEL
LIN {X 0,Y 608.414,Z 279.693,A -85,B 0,C 180,E1 -327.902,E2 -327.902} C_VEL
LIN {X 0,Y 608.395,Z 279.694,A -85,B 0,C 180,E1 -330.216,E2 -330.216} C_VEL
LIN {X 0,Y 608.391,Z 279.694,A -85,B 0,C 180,E1 -332.479,E2 -332.479} C_VEL
LIN {X 0,Y 608.421,Z 279.7,A -85,B 0,C 180,E1 -335.427,E2 -335.427} C_VEL
LIN {X 0,Y 608.411,Z 279.693,A -85,B 0,C 180,E1 -338.306,E2 -338.306} C_VEL
LIN {X 0,Y 608.393,Z 279.695,A -85,B 0,C 180,E1 -340.427,E2 -340.427} C_VEL
LIN {X 0,Y 608.402,Z 279.695,A -85,B 0,C 180,E1 -343.214,E2 -343.214} C_VEL
LIN {X 0,Y 608.466,Z 279.695,A -85,B 0,C 180,E1 -345.98,E2 -345.98} C_VEL
LIN {X 0,Y 608.402,Z 279.694,A -85,B 0,C 180,E1 -348.675,E2 -348.675} C_VEL
LIN {X 0,Y 608.418,Z 279.692,A -85,B 0,C 180,E1 -350.693,E2 -350.693} C_VEL
LIN {X 0,Y 608.407,Z 279.694,A -85,B 0,C 180,E1 -352.7,E2 -352.7} C_VEL
LIN {X 0,Y 608.421,Z 279.693,A -85,B 0,C 180,E1 -354.698,E2 -354.698} C_VEL
LIN {X 0,Y 608.413,Z 279.691,A -85,B 0,C 180,E1 -357.352,E2 -357.352} C_VEL
LIN {X 0,Y 608.444,Z 279.693,A -85,B 0,C 180,E1 -360,E2 -360} C_VEL
LIN {X 0,Y 608.478,Z 279.69,A -85,B 0,C 180,E1 -362.648,E2 -362.648} C_VEL
LIN {X 0,Y 608.413,Z 279.692,A -85,B 0,C 180,E1 -365.302,E2 -365.302} C_VEL
LIN {X 0,Y 608.411,Z 279.692,A -85,B 0,C 180,E1 -367.3,E2 -367.3} C_VEL
LIN {X 0,Y 608.433,Z 279.69,A -85,B 0,C 180,E1 -369.306,E2 -369.306} C_VEL
LIN {X 0,Y 608.421,Z 279.692,A -85,B 0,C 180,E1 -371.325,E2 -371.325} C_VEL
LIN {X 0,Y 608.437,Z 279.69,A -85,B 0,C 180,E1 -373.357,E2 -373.357} C_VEL
LIN {X 0,Y 608.45,Z 279.689,A -85,B 0,C 180,E1 -375.406,E2 -375.406} C_VEL
LIN {X 0,Y 608.401,Z 279.693,A -85,B 0,C 180,E1 -378.173,E2 -378.173} C_VEL
LIN {X 0,Y 608.442,Z 279.699,A -85,B 0,C 180,E1 -380.982,E2 -380.982} C_VEL
LIN {X 0,Y 608.432,Z 279.69,A -85,B 0,C 180,E1 -383.846,E2 -383.846} C_VEL
LIN {X 0,Y 608.414,Z 279.691,A -85,B 0,C 180,E1 -386.037,E2 -386.037} C_VEL
LIN {X 0,Y 608.407,Z 279.692,A -85,B 0,C 180,E1 -388.269,E2 -388.269} C_VEL
LIN {X 0,Y 608.418,Z 279.691,A -85,B 0,C 180,E1 -390.548,E2 -390.548} C_VEL
LIN {X 0,Y 608.435,Z 279.691,A -85,B 0,C 180,E1 -392.881,E2 -392.881} C_VEL
LIN {X 0,Y 608.431,Z 279.697,A -85,B 0,C 180,E1 -395.279,E2 -395.279} C_VEL
LIN {X 0,Y 608.455,Z 279.687,A -85,B 0,C 180,E1 -398.24,E2 -398.24} C_VEL
LIN {X 0,Y 608.42,Z 279.694,A -85,B 0,C 180,E1 -401.18,E2 -401.18} C_VEL
LIN {X 0,Y 608.472,Z 279.693,A -85,B 0,C 180,E1 -403.869,E2 -403.869} C_VEL
LIN {X 0,Y 608.445,Z 279.687,A -85,B 0,C 180,E1 -406.694,E2 -406.694} C_VEL
LIN {X 0,Y 608.426,Z 279.69,A -85,B 0,C 180,E1 -408.822,E2 -408.822} C_VEL
LIN {X 0,Y 608.457,Z 279.693,A -85,B 0,C 180,E1 -411.761,E2 -411.761} C_VEL
LIN {X 0,Y 608.434,Z 279.69,A -85,B 0,C 180,E1 -414.723,E2 -414.723} C_VEL
LIN {X 0,Y 608.444,Z 279.687,A -85,B 0,C 180,E1 -417.121,E2 -417.121} C_VEL
LIN {X 0,Y 608.432,Z 279.689,A -85,B 0,C 180,E1 -419.454,E2 -419.454} C_VEL
LIN {X 0,Y 608.424,Z 279.692,A -85,B 0,C 180,E1 -421.733,E2 -421.733} C_VEL
LIN {X 0,Y 608.475,Z 279.693,A -85,B 0,C 180,E1 -424.279,E2 -424.279} C_VEL
LIN {X 0,Y 608.449,Z 279.692,A -85,B 0,C 180,E1 -426.877,E2 -426.877} C_VEL
LIN {X 0,Y 608.461,Z 279.896,A -85,B 0,C 180,E1 -427.729,E2 -427.729} C_VEL
LIN {X 0,Y 608.558,Z 296.582,A -85,B 0,C 180,E1 -430.082,E2 -430.082} C_VEL
LIN {X 0,Y 608.499,Z 317.99,A -85,B 0,C 180,E1 -433.045,E2 -433.045} C_VEL
LIN {X 0,Y 608.474,Z 338.139,A -85,B 0,C 180,E1 -435.793,E2 -435.793} C_VEL
LIN {X 0,Y 608.512,Z 347.195,A -85,B 0,C 180,E1 -436.985,E2 -436.985} C_VEL
LIN {X 0,Y 608.541,Z 454.98,A -85,B 0,C 180,E1 -438.277,E2 -438.277} C_VEL
LIN {X 0,Y 608.543,Z 468.238,A -85,B 0,C 180,E1 -438.573,E2 -438.573} C_VEL
LIN {X 0,Y 608.517,Z 480.601,A -85,B 0,C 180,E1 -438.981,E2 -438.981} C_VEL
LIN {X 0,Y 608.512,Z 492.646,A -85,B 0,C 180,E1 -439.52,E2 -439.52} C_VEL
LIN {X 0,Y 608.467,Z 504.206,A -85,B 0,C 180,E1 -440.191,E2 -440.191} C_VEL
LIN {X 0,Y 608.472,Z 513.486,A -85,B 0,C 180,E1 -440.862,E2 -440.862} C_VEL
LIN {X 0,Y 608.487,Z 521.309,A -85,B 0,C 180,E1 -441.532,E2 -441.532} C_VEL
LIN {X 0,Y 608.47,Z 530.965,A -85,B 0,C 180,E1 -442.534,E2 -442.534} C_VEL
LIN {X 0,Y 608.435,Z 538.303,A -85,B 0,C 180,E1 -443.487,E2 -443.487} C_VEL
LIN {X 0,Y 608.45,Z 543.869,A -85,B 0,C 180,E1 -444.366,E2 -444.366} C_VEL
LIN {X 0,Y 608.432,Z 548.952,A -85,B 0,C 180,E1 -445.363,E2 -445.363} C_VEL
LIN {X 0,Y 608.449,Z 552.898,A -85,B 0,C 180,E1 -446.358,E2 -446.358} C_VEL
LIN {X 0,Y 608.425,Z 555.81,A -85,B 0,C 180,E1 -447.352,E2 -447.352} C_VEL
LIN {X 0,Y 608.441,Z 557.202,A -85,B 0,C 180,E1 -448.015,E2 -448.015} C_VEL
LIN {X 0,Y 608.438,Z 558.784,A -85,B 0,C 180,E1 -449.339,E2 -449.339} C_VEL
LIN {X 0,Y 608.434,Z 559,A -85,B 0,C 180,E1 -450,E2 -450} C_VEL
LIN {X 0,Y 608.448,Z 558.183,A -85,B 0,C 180,E1 -451.324,E2 -451.324} C_VEL
LIN {X 0,Y 608.441,Z 557.201,A -85,B 0,C 180,E1 -451.986,E2 -451.986} C_VEL
LIN {X 0,Y 608.425,Z 555.808,A -85,B 0,C 180,E1 -452.649,E2 -452.649} C_VEL
LIN {X 0,Y 608.449,Z 552.895,A -85,B 0,C 180,E1 -453.643,E2 -453.643} C_VEL
LIN {X 0,Y 608.432,Z 548.948,A -85,B 0,C 180,E1 -454.638,E2 -454.638} C_VEL
LIN {X 0,Y 608.437,Z 542.874,A -85,B 0,C 180,E1 -455.801,E2 -455.801} C_VEL
LIN {X 0,Y 608.461,Z 536.232,A -85,B 0,C 180,E1 -456.8,E2 -456.8} C_VEL
LIN {X 0,Y 608.456,Z 527.985,A -85,B 0,C 180,E1 -457.801,E2 -457.801} C_VEL
LIN {X 0,Y 608.469,Z 518.542,A -85,B 0,C 180,E1 -458.72,E2 -458.72} C_VEL
LIN {X 0,Y 608.479,Z 507.924,A -85,B 0,C 180,E1 -459.558,E2 -459.558} C_VEL
LIN {X 0,Y 608.479,Z 497.321,A -85,B 0,C 180,E1 -460.229,E2 -460.229} C_VEL
LIN {X 0,Y 608.512,Z 485.128,A -85,B 0,C 180,E1 -460.832,E2 -460.832} C_VEL
LIN {X 0,Y 608.534,Z 472.87,A -85,B 0,C 180,E1 -461.29,E2 -461.29} C_VEL
LIN {X 0,Y 608.553,Z 460.508,A -85,B 0,C 180,E1 -461.618,E2 -461.618} C_VEL
LIN {X 0,Y 608.558,Z 447.278,A -85,B 0,C 180,E1 -461.829,E2 -461.829} C_VEL
LIN {X 0,Y 608.475,Z 347.112,A -85,B 0,C 180,E1 -463.017,E2 -463.017} C_VEL
LIN {X 0,Y 608.503,Z 326.798,A -85,B 0,C 180,E1 -465.749,E2 -465.749} C_VEL
LIN {X 0,Y 608.506,Z 306.805,A -85,B 0,C 180,E1 -468.497,E2 -468.497} C_VEL
LIN {X 0,Y 608.567,Z 287.759,A -85,B 0,C 180,E1 -471.155,E2 -471.155} C_VEL
LIN {X 0,Y 608.431,Z 279.691,A -85,B 0,C 180,E1 -472.318,E2 -472.318} C_VEL
LIN {X 0,Y 608.441,Z 279.688,A -85,B 0,C 180,E1 -474.572,E2 -474.572} C_VEL
LIN {X 0,Y 608.486,Z 279.685,A -85,B 0,C 180,E1 -477.208,E2 -477.208} C_VEL
LIN {X 0,Y 608.451,Z 279.695,A -85,B 0,C 180,E1 -479.968,E2 -479.968} C_VEL
LIN {X 0,Y 608.436,Z 279.69,A -85,B 0,C 180,E1 -482.518,E2 -482.518} C_VEL
LIN {X 0,Y 608.425,Z 279.69,A -85,B 0,C 180,E1 -484.902,E2 -484.902} C_VEL
LIN {X 0,Y 608.47,Z 279.689,A -85,B 0,C 180,E1 -487.746,E2 -487.746} C_VEL
LIN {X 0,Y 608.445,Z 279.696,A -85,B 0,C 180,E1 -490.328,E2 -490.328} C_VEL
LIN {X 0,Y 608.424,Z 279.691,A -85,B 0,C 180,E1 -492.962,E2 -492.962} C_VEL
LIN {X 0,Y 608.46,Z 279.686,A -85,B 0,C 180,E1 -495.736,E2 -495.736} C_VEL
LIN {X 0,Y 608.456,Z 279.695,A -85,B 0,C 180,E1 -498.659,E2 -498.659} C_VEL
LIN {X 0,Y 608.458,Z 279.685,A -85,B 0,C 180,E1 -501.761,E2 -501.761} C_VEL
LIN {X 0,Y 608.447,Z 279.687,A -85,B 0,C 180,E1 -503.954,E2 -503.954} C_VEL
LIN {X 0,Y 608.467,Z 279.688,A -85,B 0,C 180,E1 -506.329,E2 -506.329} C_VEL
LIN {X 0,Y 608.462,Z 279.693,A -85,B 0,C 180,E1 -508.73,E2 -508.73} C_VEL
LIN {X 0,Y 608.451,Z 279.691,A -85,B 0,C 180,E1 -511.384,E2 -511.384} C_VEL
LIN {X 0,Y 608.427,Z 279.689,A -85,B 0,C 180,E1 -513.964,E2 -513.964} C_VEL
LIN {X 0,Y 608.452,Z 279.692,A -85,B 0,C 180,E1 -516.876,E2 -516.876} C_VEL
LIN {X 0,Y 608.441,Z 279.692,A -85,B 0,C 180,E1 -519.725,E2 -519.725} C_VEL
LIN {X 0,Y 608.427,Z 279.693,A -85,B 0,C 180,E1 -521.827,E2 -521.827} C_VEL
LIN {X 0,Y 608.438,Z 279.692,A -85,B 0,C 180,E1 -523.906,E2 -523.906} C_VEL
LIN {X 0,Y 608.431,Z 279.693,A -85,B 0,C 180,E1 -525.997,E2 -525.997} C_VEL
LIN {X 0,Y 608.441,Z 279.692,A -85,B 0,C 180,E1 -528,E2 -528} C_VEL
LIN {X 0,Y 608.448,Z 279.686,A -85,B 0,C 180,E1 -530.694,E2 -530.694} C_VEL
LIN {X 0,Y 608.479,Z 279.686,A -85,B 0,C 180,E1 -533.368,E2 -533.368} C_VEL
LIN {X 0,Y 608.452,Z 279.696,A -85,B 0,C 180,E1 -536.026,E2 -536.026} C_VEL
LIN {X 0,Y 608.439,Z 279.689,A -85,B 0,C 180,E1 -538.676,E2 -538.676} C_VEL
LIN {X 0,Y 608.457,Z 279.686,A -85,B 0,C 180,E1 -541.324,E2 -541.324} C_VEL
LIN {X 0,Y 608.459,Z 279.692,A -85,B 0,C 180,E1 -543.974,E2 -543.974} C_VEL
LIN {X 0,Y 608.438,Z 279.694,A -85,B 0,C 180,E1 -546.633,E2 -546.633} C_VEL
LIN {X 0,Y 608.446,Z 279.694,A -85,B 0,C 180,E1 -548.636,E2 -548.636} C_VEL
LIN {X 0,Y 608.441,Z 279.687,A -85,B 0,C 180,E1 -549.447,E2 -549.447} C_VEL
LIN {X 0,Y 607.781,Z 279.774,A -85,B 0,C 180,E1 -550,E2 -550} C_VEL
LIN {X 0,Y 604.937,Z 280.129,A -85,B 0,C 180,E1 -550.897,E2 -550.897} C_VEL
LIN {X 0,Y 602.529,Z 280.428,A -85,B 0,C 180,E1 -551.618,E2 -551.618} C_VEL
LIN {X 0,Y 601.492,Z 280.558,A -85,B 0,C 180,E1 -552.175,E2 -552.175} C_VEL
LIN {X 0,Y 601.405,Z 280.568,A -85,B 0,C 180,E1 -552.363,E2 -552.363} C_VEL
LIN {X 0,Y 601.42,Z 280.569,A -85,B 0,C 180,E1 -554.897,E2 -554.897} C_VEL
LIN {X 0,Y 601.424,Z 280.568,A -85,B 0,C 180,E1 -556.986,E2 -556.986} C_VEL
LIN {X 0,Y 601.391,Z 280.566,A -85,B 0,C 180,E1 -559.81,E2 -559.81} C_VEL
LIN {X 0,Y 601.401,Z 280.564,A -85,B 0,C 180,E1 -561.96,E2 -561.96} C_VEL
LIN {X 0,Y 601.398,Z 280.574,A -85,B 0,C 180,E1 -564.879,E2 -564.879} C_VEL
LIN {X 0,Y 601.401,Z 280.572,A -85,B 0,C 180,E1 -567.36,E2 -567.36} C_VEL
LIN {X 0,Y 601.403,Z 280.572,A -85,B 0,C 180,E1 -569.394,E2 -569.394} C_VEL
LIN {X 0,Y 601.39,Z 280.57,A -85,B 0,C 180,E1 -571.728,E2 -571.728} C_VEL
LIN {X 0,Y 601.416,Z 280.563,A -85,B 0,C 180,E1 -574.12,E2 -574.12} C_VEL
LIN {X 0,Y 601.4,Z 280.565,A -85,B 0,C 180,E1 -576.584,E2 -576.584} C_VEL
LIN {X 0,Y 601.438,Z 280.571,A -85,B 0,C 180,E1 -579.535,E2 -579.535} C_VEL
LIN {X 0,Y 601.414,Z 280.573,A -85,B 0,C 180,E1 -581.766,E2 -581.766} C_VEL
LIN {X 0,Y 601.401,Z 280.565,A -85,B 0,C 180,E1 -584.533,E2 -584.533} C_VEL
LIN {X 0,Y 601.412,Z 280.567,A -85,B 0,C 180,E1 -587.41,E2 -587.41} C_VEL
LIN {X 0,Y 601.401,Z 280.577,A -85,B 0,C 180,E1 -590.004,E2 -590.004} C_VEL
LIN {X 0,Y 601.401,Z 280.568,A -85,B 0,C 180,E1 -592.623,E2 -592.623} C_VEL
LIN {X 0,Y 601.386,Z 280.567,A -85,B 0,C 180,E1 -595.066,E2 -595.066} C_VEL
LIN {X 0,Y 601.422,Z 280.563,A -85,B 0,C 180,E1 -597.484,E2 -597.484} C_VEL
LIN {X 0,Y 601.443,Z 280.674,A -85,B 0,C 180,E1 -599.643,E2 -599.643} C_VEL
LIN {X 0,Y 601.495,Z 295.502,A -85,B 0,C 180,E1 -602.136,E2 -602.136} C_VEL
LIN {X 0,Y 601.458,Z 312.426,A -85,B 0,C 180,E1 -604.939,E2 -604.939} C_VEL
LIN {X 0,Y 601.428,Z 318.165,A -85,B 0,C 180,E1 -605.881,E2 -605.881} C_VEL
LIN {X 0,Y 601.7,Z 323.961,A -85,B 0,C 180,E1 -605.961,E2 -605.961} C_VEL
LIN {X 0,Y 601.593,Z 425.144,A -85,B 0,C 180,E1 -607.188,E2 -607.188} C_VEL
LIN {X 0,Y 601.572,Z 438.405,A -85,B 0,C 180,E1 -607.488,E2 -607.488} C_VEL
LIN {X 0,Y 601.568,Z 451.036,A -85,B 0,C 180,E1 -607.914,E2 -607.914} C_VEL
LIN {X 0,Y 601.479,Z 463.621,A -85,B 0,C 180,E1 -608.494,E2 -608.494} C_VEL
LIN {X 0,Y 601.466,Z 475.31,A -85,B 0,C 180,E1 -609.194,E2 -609.194} C_VEL
LIN {X 0,Y 601.455,Z 484.997,A -85,B 0,C 180,E1 -609.925,E2 -609.925} C_VEL
LIN {X 0,Y 601.446,Z 492.022,A -85,B 0,C 180,E1 -610.547,E2 -610.547} C_VEL
LIN {X 0,Y 601.396,Z 500.142,A -85,B 0,C 180,E1 -611.397,E2 -611.397} C_VEL
LIN {X 0,Y 601.38,Z 507.303,A -85,B 0,C 180,E1 -612.311,E2 -612.311} C_VEL
LIN {X 0,Y 601.347,Z 514.198,A -85,B 0,C 180,E1 -613.405,E2 -613.405} C_VEL
LIN {X 0,Y 601.338,Z 519.179,A -85,B 0,C 180,E1 -614.406,E2 -614.406} C_VEL
LIN {X 0,Y 601.327,Z 523.173,A -85,B 0,C 180,E1 -615.446,E2 -615.446} C_VEL
LIN {X 0,Y 601.341,Z 526.073,A -85,B 0,C 180,E1 -616.482,E2 -616.482} C_VEL
LIN {X 0,Y 601.325,Z 527.422,A -85,B 0,C 180,E1 -617.169,E2 -617.169} C_VEL
LIN {X 0,Y 601.342,Z 528.359,A -85,B 0,C 180,E1 -617.856,E2 -617.856} C_VEL
LIN {X 0,Y 601.351,Z 528.999,A -85,B 0,C 180,E1 -619.027,E2 -619.027} C_VEL
LIN {X 0,Y 601.328,Z 528.653,A -85,B 0,C 180,E1 -619.903,E2 -619.903} C_VEL
LIN {X 0,Y 601.337,Z 527.952,A -85,B 0,C 180,E1 -620.582,E2 -620.582} C_VEL
LIN {X 0,Y 601.333,Z 526.815,A -85,B 0,C 180,E1 -621.26,E2 -621.26} C_VEL
LIN {X 0,Y 601.333,Z 525.249,A -85,B 0,C 180,E1 -621.937,E2 -621.937} C_VEL
LIN {X 0,Y 601.366,Z 522.099,A -85,B 0,C 180,E1 -622.951,E2 -622.951} C_VEL
LIN {X 0,Y 601.357,Z 517.901,A -85,B 0,C 180,E1 -623.962,E2 -623.962} C_VEL
LIN {X 0,Y 601.392,Z 511.524,A -85,B 0,C 180,E1 -625.139,E2 -625.139} C_VEL
LIN {X 0,Y 601.377,Z 504.606,A -85,B 0,C 180,E1 -626.147,E2 -626.147} C_VEL
LIN {X 0,Y 601.428,Z 495.942,A -85,B 0,C 180,E1 -627.153,E2 -627.153} C_VEL
LIN {X 0,Y 601.441,Z 487.087,A -85,B 0,C 180,E1 -627.991,E2 -627.991} C_VEL
LIN {X 0,Y 601.455,Z 477.528,A -85,B 0,C 180,E1 -628.744,E2 -628.744} C_VEL
LIN {X 0,Y 601.485,Z 466.981,A -85,B 0,C 180,E1 -629.414,E2 -629.414} C_VEL
LIN {X 0,Y 601.55,Z 455.24,A -85,B 0,C 180,E1 -630,E2 -630} C_VEL
LIN {X 0,Y 601.549,Z 443.131,A -85,B 0,C 180,E1 -630.46,E2 -630.46} C_VEL
LIN {X 0,Y 601.561,Z 430.747,A -85,B 0,C 180,E1 -630.794,E2 -630.794} C_VEL
LIN {X 0,Y 601.6,Z 418.065,A -85,B 0,C 180,E1 -631.004,E2 -631.004} C_VEL
LIN {X 0,Y 601.607,Z 319.371,A -85,B 0,C 180,E1 -632.186,E2 -632.186} C_VEL
LIN {X 0,Y 601.427,Z 318.111,A -85,B 0,C 180,E1 -632.218,E2 -632.218} C_VEL
LIN {X 0,Y 601.44,Z 302.091,A -85,B 0,C 180,E1 -634.859,E2 -634.859} C_VEL
LIN {X 0,Y 601.52,Z 285.958,A -85,B 0,C 180,E1 -637.552,E2 -637.552} C_VEL
LIN {X 0,Y 601.397,Z 280.569,A -85,B 0,C 180,E1 -638.484,E2 -638.484} C_VEL
LIN {X 0,Y 601.401,Z 280.565,A -85,B 0,C 180,E1 -640.998,E2 -640.998} C_VEL
LIN {X 0,Y 601.419,Z 280.571,A -85,B 0,C 180,E1 -644.089,E2 -644.089} C_VEL
LIN {X 0,Y 601.374,Z 280.568,A -85,B 0,C 180,E1 -646.987,E2 -646.987} C_VEL
LIN {X 0,Y 601.391,Z 280.572,A -85,B 0,C 180,E1 -649.809,E2 -649.809} C_VEL
LIN {X 0,Y 601.398,Z 280.568,A -85,B 0,C 180,E1 -652.683,E2 -652.683} C_VEL
LIN {X 0,Y 601.372,Z 280.57,A -85,B 0,C 180,E1 -654.879,E2 -654.879} C_VEL
LIN {X 0,Y 601.367,Z 280.569,A -85,B 0,C 180,E1 -657.353,E2 -657.353} C_VEL
LIN {X 0,Y 601.404,Z 280.571,A -85,B 0,C 180,E1 -660.164,E2 -660.164} C_VEL
LIN {X 0,Y 601.414,Z 280.571,A -85,B 0,C 180,E1 -662.713,E2 -662.713} C_VEL
LIN {X 0,Y 601.366,Z 280.572,A -85,B 0,C 180,E1 -665.107,E2 -665.107} C_VEL
LIN {X 0,Y 601.379,Z 280.568,A -85,B 0,C 180,E1 -667.422,E2 -667.422} C_VEL
LIN {X 0,Y 601.379,Z 280.568,A -85,B 0,C 180,E1 -669.996,E2 -669.996} C_VEL
LIN {X 0,Y 601.374,Z 280.577,A -85,B 0,C 180,E1 -672.672,E2 -672.672} C_VEL
LIN {X 0,Y 601.363,Z 280.572,A -85,B 0,C 180,E1 -675.476,E2 -675.476} C_VEL
LIN {X 0,Y 601.397,Z 280.567,A -85,B 0,C 180,E1 -678.408,E2 -678.408} C_VEL
LIN {X 0,Y 601.386,Z 280.571,A -85,B 0,C 180,E1 -681.533,E2 -681.533} C_VEL
LIN {X 0,Y 601.347,Z 280.571,A -85,B 0,C 180,E1 -684.242,E2 -684.242} C_VEL
LIN {X 0,Y 601.361,Z 280.572,A -85,B 0,C 180,E1 -686.682,E2 -686.682} C_VEL
LIN {X 0,Y 601.369,Z 280.575,A -85,B 0,C 180,E1 -689.055,E2 -689.055} C_VEL
LIN {X 0,Y 601.416,Z 280.574,A -85,B 0,C 180,E1 -691.372,E2 -691.372} C_VEL
LIN {X 0,Y 601.352,Z 280.571,A -85,B 0,C 180,E1 -694.379,E2 -694.379} C_VEL
LIN {X 0,Y 601.341,Z 280.572,A -85,B 0,C 180,E1 -696.586,E2 -696.586} C_VEL
LIN {X 0,Y 601.383,Z 280.57,A -85,B 0,C 180,E1 -699.211,E2 -699.211} C_VEL
LIN {X 0,Y 601.367,Z 280.578,A -85,B 0,C 180,E1 -701.606,E2 -701.606} C_VEL
LIN {X 0,Y 601.366,Z 280.571,A -85,B 0,C 180,E1 -704.407,E2 -704.407} C_VEL
LIN {X 0,Y 601.374,Z 280.57,A -85,B 0,C 180,E1 -706.483,E2 -706.483} C_VEL
LIN {X 0,Y 601.364,Z 280.569,A -85,B 0,C 180,E1 -709.013,E2 -709.013} C_VEL
LIN {X 0,Y 601.363,Z 280.57,A -85,B 0,C 180,E1 -711.261,E2 -711.261} C_VEL
LIN {X 0,Y 601.403,Z 280.573,A -85,B 0,C 180,E1 -713.963,E2 -713.963} C_VEL
LIN {X 0,Y 601.397,Z 280.569,A -85,B 0,C 180,E1 -716.65,E2 -716.65} C_VEL
LIN {X 0,Y 601.351,Z 280.571,A -85,B 0,C 180,E1 -719.33,E2 -719.33} C_VEL
LIN {X 0,Y 601.365,Z 280.569,A -85,B 0,C 180,E1 -721.339,E2 -721.339} C_VEL
LIN {X 0,Y 601.348,Z 280.571,A -85,B 0,C 180,E1 -723.35,E2 -723.35} C_VEL
LIN {X 0,Y 601.378,Z 280.568,A -85,B 0,C 180,E1 -725.364,E2 -725.364} C_VEL
LIN {X 0,Y 601.36,Z 280.57,A -85,B 0,C 180,E1 -727.386,E2 -727.386} C_VEL
LIN {X 0,Y 601.378,Z 280.568,A -85,B 0,C 180,E1 -729.416,E2 -729.416} C_VEL
LIN {X 0,Y 601.392,Z 280.566,A -85,B 0,C 180,E1 -731.459,E2 -731.459} C_VEL
LIN {X 0,Y 601.39,Z 280.568,A -85,B 0,C 180,E1 -734.206,E2 -734.206} C_VEL
LIN {X 0,Y 601.401,Z 280.574,A -85,B 0,C 180,E1 -736.987,E2 -736.987} C_VEL
LIN {X 0,Y 601.377,Z 280.568,A -85,B 0,C 180,E1 -739.81,E2 -739.81} C_VEL
LIN {X 0,Y 601.393,Z 280.57,A -85,B 0,C 180,E1 -742.684,E2 -742.684} C_VEL
LIN {X 0,Y 601.425,Z 280.565,A -85,B 0,C 180,E1 -745.618,E2 -745.618} C_VEL
LIN {X 0,Y 601.379,Z 280.569,A -85,B 0,C 180,E1 -747.87,E2 -747.87} C_VEL
LIN {X 0,Y 601.392,Z 280.566,A -85,B 0,C 180,E1 -750.166,E2 -750.166} C_VEL
LIN {X 0,Y 601.391,Z 280.567,A -85,B 0,C 180,E1 -752.713,E2 -752.713} C_VEL
LIN {X 0,Y 601.374,Z 280.573,A -85,B 0,C 180,E1 -755.111,E2 -755.111} C_VEL
LIN {X 0,Y 601.424,Z 280.571,A -85,B 0,C 180,E1 -757.42,E2 -757.42} C_VEL
LIN {X 0,Y 601.395,Z 280.57,A -85,B 0,C 180,E1 -759.996,E2 -759.996} C_VEL
LIN {X 0,Y 601.372,Z 280.568,A -85,B 0,C 180,E1 -762.674,E2 -762.674} C_VEL
LIN {X 0,Y 601.392,Z 280.566,A -85,B 0,C 180,E1 -764.533,E2 -764.533} C_VEL
LIN {X 0,Y 601.422,Z 280.564,A -85,B 0,C 180,E1 -766.428,E2 -766.428} C_VEL
LIN {X 0,Y 601.395,Z 280.566,A -85,B 0,C 180,E1 -769.125,E2 -769.125} C_VEL
LIN {X 0,Y 601.408,Z 280.571,A -85,B 0,C 180,E1 -771.732,E2 -771.732} C_VEL
LIN {X 0,Y 601.384,Z 280.575,A -85,B 0,C 180,E1 -774.246,E2 -774.246} C_VEL
LIN {X 0,Y 601.422,Z 280.565,A -85,B 0,C 180,E1 -776.687,E2 -776.687} C_VEL
LIN {X 0,Y 601.415,Z 280.563,A -85,B 0,C 180,E1 -779.059,E2 -779.059} C_VEL
LIN {X 0,Y 601.406,Z 280.564,A -85,B 0,C 180,E1 -781.373,E2 -781.373} C_VEL
LIN {X 0,Y 601.392,Z 280.567,A -85,B 0,C 180,E1 -783.637,E2 -783.637} C_VEL
LIN {X 0,Y 601.413,Z 280.574,A -85,B 0,C 180,E1 -786.59,E2 -786.59} C_VEL
LIN {X 0,Y 601.42,Z 280.588,A -85,B 0,C 180,E1 -787.554,E2 -787.554} C_VEL
LIN {X 0,Y 601.624,Z 290.948,A -85,B 0,C 180,E1 -789.043,E2 -789.043} C_VEL
LIN {X 0,Y 601.521,Z 310.434,A -85,B 0,C 180,E1 -791.788,E2 -791.788} C_VEL
LIN {X 0,Y 601.51,Z 329.324,A -85,B 0,C 180,E1 -794.412,E2 -794.412} C_VEL
LIN {X 0,Y 601.45,Z 347.195,A -85,B 0,C 180,E1 -796.83,E2 -796.83} C_VEL
LIN {X 0,Y 601.659,Z 374.025,A -85,B 0,C 180,E1 -797.156,E2 -797.156} C_VEL
LIN {X 0,Y 601.611,Z 454.98,A -85,B 0,C 180,E1 -798.14,E2 -798.14} C_VEL
LIN {X 0,Y 601.586,Z 468.239,A -85,B 0,C 180,E1 -798.439,E2 -798.439} C_VEL
LIN {X 0,Y 601.544,Z 479.978,A -85,B 0,C 180,E1 -798.828,E2 -798.828} C_VEL
LIN {X 0,Y 601.528,Z 490.936,A -85,B 0,C 180,E1 -799.312,E2 -799.312} C_VEL
LIN {X 0,Y 601.457,Z 501.59,A -85,B 0,C 180,E1 -799.906,E2 -799.906} C_VEL
LIN {X 0,Y 601.445,Z 512.483,A -85,B 0,C 180,E1 -800.67,E2 -800.67} C_VEL
LIN {X 0,Y 601.423,Z 521.323,A -85,B 0,C 180,E1 -801.432,E2 -801.432} C_VEL
LIN {X 0,Y 601.396,Z 529.483,A -85,B 0,C 180,E1 -802.277,E2 -802.277} C_VEL
LIN {X 0,Y 601.381,Z 537.474,A -85,B 0,C 180,E1 -803.289,E2 -803.289} C_VEL
LIN {X 0,Y 601.371,Z 543.869,A -85,B 0,C 180,E1 -804.3,E2 -804.3} C_VEL
LIN {X 0,Y 601.336,Z 548.952,A -85,B 0,C 180,E1 -805.308,E2 -805.308} C_VEL
LIN {X 0,Y 601.367,Z 552.898,A -85,B 0,C 180,E1 -806.315,E2 -806.315} C_VEL
LIN {X 0,Y 601.325,Z 555.81,A -85,B 0,C 180,E1 -807.321,E2 -807.321} C_VEL
LIN {X 0,Y 601.34,Z 557.203,A -85,B 0,C 180,E1 -807.991,E2 -807.991} C_VEL
LIN {X 0,Y 601.339,Z 558.784,A -85,B 0,C 180,E1 -809.331,E2 -809.331} C_VEL
LIN {X 0,Y 601.335,Z 559,A -85,B 0,C 180,E1 -810,E2 -810} C_VEL
LIN {X 0,Y 601.348,Z 558.184,A -85,B 0,C 180,E1 -811.34,E2 -811.34} C_VEL
LIN {X 0,Y 601.34,Z 557.201,A -85,B 0,C 180,E1 -812.01,E2 -812.01} C_VEL
LIN {X 0,Y 601.325,Z 555.808,A -85,B 0,C 180,E1 -812.68,E2 -812.68} C_VEL
LIN {X 0,Y 601.367,Z 552.895,A -85,B 0,C 180,E1 -813.686,E2 -813.686} C_VEL
LIN {X 0,Y 601.336,Z 548.948,A -85,B 0,C 180,E1 -814.693,E2 -814.693} C_VEL
LIN {X 0,Y 601.372,Z 542.874,A -85,B 0,C 180,E1 -815.87,E2 -815.87} C_VEL
LIN {X 0,Y 601.381,Z 536.232,A -85,B 0,C 180,E1 -816.88,E2 -816.88} C_VEL
LIN {X 0,Y 601.4,Z 527.986,A -85,B 0,C 180,E1 -817.893,E2 -817.893} C_VEL
LIN {X 0,Y 601.433,Z 519.532,A -85,B 0,C 180,E1 -818.738,E2 -818.738} C_VEL
LIN {X 0,Y 601.44,Z 509.087,A -85,B 0,C 180,E1 -819.586,E2 -819.586} C_VEL
LIN {X 0,Y 601.472,Z 498.751,A -85,B 0,C 180,E1 -820.265,E2 -820.265} C_VEL
LIN {X 0,Y 601.539,Z 486.574,A -85,B 0,C 180,E1 -820.897,E2 -820.897} C_VEL
LIN {X 0,Y 601.569,Z 474.203,A -85,B 0,C 180,E1 -821.379,E2 -821.379} C_VEL
LIN {X 0,Y 601.586,Z 461.421,A -85,B 0,C 180,E1 -821.733,E2 -821.733} C_VEL
LIN {X 0,Y 601.616,Z 449.055,A -85,B 0,C 180,E1 -821.946,E2 -821.946} C_VEL
LIN {X 0,Y 601.553,Z 347.782,A -85,B 0,C 180,E1 -823.161,E2 -823.161} C_VEL
LIN {X 0,Y 601.445,Z 346.79,A -85,B 0,C 180,E1 -823.193,E2 -823.193} C_VEL
LIN {X 0,Y 601.507,Z 326.798,A -85,B 0,C 180,E1 -825.937,E2 -825.937} C_VEL
LIN {X 0,Y 601.532,Z 307.493,A -85,B 0,C 180,E1 -828.623,E2 -828.623} C_VEL
LIN {X 0,Y 601.655,Z 287.759,A -85,B 0,C 180,E1 -831.41,E2 -831.41} C_VEL
LIN {X 0,Y 601.41,Z 280.568,A -85,B 0,C 180,E1 -832.469,E2 -832.469} C_VEL
LIN {X 0,Y 601.4,Z 280.566,A -85,B 0,C 180,E1 -834.879,E2 -834.879} C_VEL
LIN {X 0,Y 601.421,Z 280.568,A -85,B 0,C 180,E1 -837.363,E2 -837.363} C_VEL
LIN {X 0,Y 601.405,Z 280.57,A -85,B 0,C 180,E1 -840.166,E2 -840.166} C_VEL
LIN {X 0,Y 601.405,Z 280.565,A -85,B 0,C 180,E1 -842.713,E2 -842.713} C_VEL
LIN {X 0,Y 601.383,Z 280.567,A -85,B 0,C 180,E1 -845.11,E2 -845.11} C_VEL
LIN {X 0,Y 601.434,Z 280.562,A -85,B 0,C 180,E1 -847.419,E2 -847.419} C_VEL
LIN {X 0,Y 601.402,Z 280.573,A -85,B 0,C 180,E1 -849.996,E2 -849.996} C_VEL
LIN {X 0,Y 601.404,Z 280.569,A -85,B 0,C 180,E1 -852.671,E2 -852.671} C_VEL
LIN {X 0,Y 601.4,Z 280.565,A -85,B 0,C 180,E1 -855.479,E2 -855.479} C_VEL
LIN {X 0,Y 601.424,Z 280.572,A -85,B 0,C 180,E1 -858.407,E2 -858.407} C_VEL
LIN {X 0,Y 601.398,Z 280.571,A -85,B 0,C 180,E1 -860.872,E2 -860.872} C_VEL
LIN {X 0,Y 601.39,Z 280.567,A -85,B 0,C 180,E1 -863.416,E2 -863.416} C_VEL
LIN {X 0,Y 601.429,Z 280.562,A -85,B 0,C 180,E1 -866.065,E2 -866.065} C_VEL
LIN {X 0,Y 601.408,Z 280.573,A -85,B 0,C 180,E1 -869.057,E2 -869.057} C_VEL
LIN {X 0,Y 601.412,Z 280.568,A -85,B 0,C 180,E1 -871.372,E2 -871.372} C_VEL
LIN {X 0,Y 601.391,Z 280.568,A -85,B 0,C 180,E1 -873.636,E2 -873.636} C_VEL
LIN {X 0,Y 601.406,Z 280.565,A -85,B 0,C 180,E1 -875.857,E2 -875.857} C_VEL
LIN {X 0,Y 601.392,Z 280.566,A -85,B 0,C 180,E1 -878.04,E2 -878.04} C_VEL
LIN {X 0,Y 601.392,Z 280.566,A -85,B 0,C 180,E1 -880.19,E2 -880.19} C_VEL
LIN {X 0,Y 601.43,Z 280.565,A -85,B 0,C 180,E1 -883.014,E2 -883.014} C_VEL
LIN {X 0,Y 601.399,Z 280.569,A -85,B 0,C 180,E1 -885.917,E2 -885.917} C_VEL
LIN {X 0,Y 601.407,Z 280.564,A -85,B 0,C 180,E1 -888.541,E2 -888.541} C_VEL
LIN {X 0,Y 601.414,Z 280.566,A -85,B 0,C 180,E1 -891.262,E2 -891.262} C_VEL
LIN {X 0,Y 601.403,Z 280.574,A -85,B 0,C 180,E1 -893.963,E2 -893.963} C_VEL
LIN {X 0,Y 601.405,Z 280.575,A -85,B 0,C 180,E1 -895.979,E2 -895.979} C_VEL
LIN {X 0,Y 601.435,Z 280.572,A -85,B 0,C 180,E1 -897.991,E2 -897.991} C_VEL
LIN {X 0,Y 601.425,Z 280.564,A -85,B 0,C 180,E1 -900.67,E2 -900.67} C_VEL
LIN {X 0,Y 601.412,Z 280.563,A -85,B 0,C 180,E1 -903.35,E2 -903.35} C_VEL
LIN {X 0,Y 601.433,Z 280.567,A -85,B 0,C 180,E1 -906.037,E2 -906.037} C_VEL
LIN {X 0,Y 601.404,Z 280.57,A -85,B 0,C 180,E1 -908.738,E2 -908.738} C_VEL
LIN {X 0,Y 601.403,Z 280.567,A -85,B 0,C 180,E1 -911.002,E2 -911.002} C_VEL
LIN {X 0,Y 601.405,Z 280.568,A -85,B 0,C 180,E1 -912.363,E2 -912.363} C_VEL
LIN {X 0,Y 600.735,Z 280.654,A -85,B 0,C 180,E1 -912.923,E2 -912.923} C_VEL
LIN {X 0,Y 597.884,Z 281.009,A -85,B 0,C 180,E1 -913.831,E2 -913.831} C_VEL
LIN {X 0,Y 595.475,Z 281.313,A -85,B 0,C 180,E1 -914.561,E2 -914.561} C_VEL
LIN {X 0,Y 594.437,Z 281.436,A -85,B 0,C 180,E1 -915.124,E2 -915.124} C_VEL
LIN {X 0,Y 594.35,Z 281.445,A -85,B 0,C 180,E1 -915.315,E2 -915.315} C_VEL
LIN {X 0,Y 594.38,Z 281.442,A -85,B 0,C 180,E1 -917.194,E2 -917.194} C_VEL
LIN {X 0,Y 594.367,Z 281.441,A -85,B 0,C 180,E1 -920.054,E2 -920.054} C_VEL
LIN {X 0,Y 594.353,Z 281.454,A -85,B 0,C 180,E1 -922.968,E2 -922.968} C_VEL
LIN {X 0,Y 594.358,Z 281.451,A -85,B 0,C 180,E1 -925.194,E2 -925.194} C_VEL
LIN {X 0,Y 594.348,Z 281.447,A -85,B 0,C 180,E1 -927.52,E2 -927.52} C_VEL
LIN {X 0,Y 594.357,Z 281.444,A -85,B 0,C 180,E1 -929.778,E2 -929.778} C_VEL
LIN {X 0,Y 594.355,Z 281.443,A -85,B 0,C 180,E1 -932.148,E2 -932.148} C_VEL
LIN {X 0,Y 594.392,Z 281.438,A -85,B 0,C 180,E1 -934.58,E2 -934.58} C_VEL
LIN {X 0,Y 594.387,Z 281.449,A -85,B 0,C 180,E1 -937.608,E2 -937.608} C_VEL
LIN {X 0,Y 594.362,Z 281.442,A -85,B 0,C 180,E1 -940.568,E2 -940.568} C_VEL
LIN {X 0,Y 594.361,Z 281.446,A -85,B 0,C 180,E1 -943.301,E2 -943.301} C_VEL
LIN {X 0,Y 594.346,Z 281.449,A -85,B 0,C 180,E1 -946.163,E2 -946.163} C_VEL
LIN {X 0,Y 594.369,Z 281.443,A -85,B 0,C 180,E1 -948.535,E2 -948.535} C_VEL
LIN {X 0,Y 594.37,Z 281.442,A -85,B 0,C 180,E1 -951.298,E2 -951.298} C_VEL
LIN {X 0,Y 594.352,Z 281.448,A -85,B 0,C 180,E1 -953.755,E2 -953.755} C_VEL
LIN {X 0,Y 594.365,Z 281.453,A -85,B 0,C 180,E1 -956.238,E2 -956.238} C_VEL
LIN {X 0,Y 594.364,Z 281.448,A -85,B 0,C 180,E1 -958.649,E2 -958.649} C_VEL
LIN {X 0,Y 594.379,Z 281.517,A -85,B 0,C 180,E1 -959.548,E2 -959.548} C_VEL
LIN {X 0,Y 594.493,Z 293.505,A -85,B 0,C 180,E1 -961.593,E2 -961.593} C_VEL
LIN {X 0,Y 594.433,Z 311.545,A -85,B 0,C 180,E1 -964.622,E2 -964.622} C_VEL
LIN {X 0,Y 594.397,Z 318.13,A -85,B 0,C 180,E1 -965.717,E2 -965.717} C_VEL
LIN {X 0,Y 594.766,Z 322.698,A -85,B 0,C 180,E1 -965.791,E2 -965.791} C_VEL
LIN {X 0,Y 594.668,Z 424.993,A -85,B 0,C 180,E1 -967.045,E2 -967.045} C_VEL
LIN {X 0,Y 594.618,Z 438.364,A -85,B 0,C 180,E1 -967.35,E2 -967.35} C_VEL
LIN {X 0,Y 594.593,Z 450.875,A -85,B 0,C 180,E1 -967.775,E2 -967.775} C_VEL
LIN {X 0,Y 594.512,Z 462.728,A -85,B 0,C 180,E1 -968.32,E2 -968.32} C_VEL
LIN {X 0,Y 594.476,Z 474.029,A -85,B 0,C 180,E1 -968.991,E2 -968.991} C_VEL
LIN {X 0,Y 594.42,Z 484.435,A -85,B 0,C 180,E1 -969.767,E2 -969.767} C_VEL
LIN {X 0,Y 594.408,Z 492.446,A -85,B 0,C 180,E1 -970.487,E2 -970.487} C_VEL
LIN {X 0,Y 594.321,Z 500.791,A -85,B 0,C 180,E1 -971.38,E2 -971.38} C_VEL
LIN {X 0,Y 594.308,Z 508.782,A -85,B 0,C 180,E1 -972.449,E2 -972.449} C_VEL
LIN {X 0,Y 594.263,Z 515.118,A -85,B 0,C 180,E1 -973.511,E2 -973.511} C_VEL
LIN {X 0,Y 594.264,Z 520.085,A -85,B 0,C 180,E1 -974.568,E2 -974.568} C_VEL
LIN {X 0,Y 594.25,Z 523.846,A -85,B 0,C 180,E1 -975.619,E2 -975.619} C_VEL
LIN {X 0,Y 594.259,Z 525.77,A -85,B 0,C 180,E1 -976.318,E2 -976.318} C_VEL
LIN {X 0,Y 594.244,Z 527.205,A -85,B 0,C 180,E1 -977.014,E2 -977.014} C_VEL
LIN {X 0,Y 594.24,Z 528.206,A -85,B 0,C 180,E1 -977.708,E2 -977.708} C_VEL
LIN {X 0,Y 594.253,Z 528.995,A -85,B 0,C 180,E1 -978.997,E2 -978.997} C_VEL
LIN {X 0,Y 594.231,Z 528.744,A -85,B 0,C 180,E1 -979.781,E2 -979.781} C_VEL
LIN {X 0,Y 594.256,Z 528.106,A -85,B 0,C 180,E1 -980.469,E2 -980.469} C_VEL
LIN {X 0,Y 594.229,Z 527.074,A -85,B 0,C 180,E1 -981.155,E2 -981.155} C_VEL
LIN {X 0,Y 594.23,Z 525.593,A -85,B 0,C 180,E1 -981.84,E2 -981.84} C_VEL
LIN {X 0,Y 594.259,Z 522.578,A -85,B 0,C 180,E1 -982.866,E2 -982.866} C_VEL
LIN {X 0,Y 594.279,Z 518.522,A -85,B 0,C 180,E1 -983.89,E2 -983.89} C_VEL
LIN {X 0,Y 594.305,Z 512.302,A -85,B 0,C 180,E1 -985.081,E2 -985.081} C_VEL
LIN {X 0,Y 594.31,Z 505.558,A -85,B 0,C 180,E1 -986.101,E2 -986.101} C_VEL
LIN {X 0,Y 594.374,Z 497.203,A -85,B 0,C 180,E1 -987.119,E2 -987.119} C_VEL
LIN {X 0,Y 594.41,Z 488.629,A -85,B 0,C 180,E1 -987.967,E2 -987.967} C_VEL
LIN {X 0,Y 594.434,Z 478.152,A -85,B 0,C 180,E1 -988.814,E2 -988.814} C_VEL
LIN {X 0,Y 594.472,Z 467.767,A -85,B 0,C 180,E1 -989.491,E2 -989.491} C_VEL
LIN {X 0,Y 594.556,Z 456.288,A -85,B 0,C 180,E1 -990.084,E2 -990.084} C_VEL
LIN {X 0,Y 594.579,Z 443.23,A -85,B 0,C 180,E1 -990.592,E2 -990.592} C_VEL
LIN {X 0,Y 594.625,Z 429.935,A -85,B 0,C 180,E1 -990.952,E2 -990.952} C_VEL
LIN {X 0,Y 594.658,Z 414.815,A -85,B 0,C 180,E1 -991.185,E2 -991.185} C_VEL
LIN {X 0,Y 594.73,Z 320.438,A -85,B 0,C 180,E1 -992.328,E2 -992.328} C_VEL
LIN {X 0,Y 594.396,Z 318.143,A -85,B 0,C 180,E1 -992.371,E2 -992.371} C_VEL
LIN {X 0,Y 594.413,Z 302.89,A -85,B 0,C 180,E1 -994.917,E2 -994.917} C_VEL
LIN {X 0,Y 594.529,Z 286.758,A -85,B 0,C 180,E1 -997.642,E2 -997.642} C_VEL
LIN {X 0,Y 594.334,Z 281.449,A -85,B 0,C 180,E1 -998.585,E2 -998.585} C_VEL
LIN {X 0,Y 594.368,Z 281.442,A -85,B 0,C 180,E1 -1001.06,E2 -1001.06} C_VEL
LIN {X 0,Y 594.375,Z 281.448,A -85,B 0,C 180,E1 -1003.678,E2 -1003.678} C_VEL
LIN {X 0,Y 594.331,Z 281.446,A -85,B 0,C 180,E1 -1006.697,E2 -1006.697} C_VEL
LIN {X 0,Y 594.356,Z 281.443,A -85,B 0,C 180,E1 -1009.334,E2 -1009.334} C_VEL
LIN {X 0,Y 594.346,Z 281.445,A -85,B 0,C 180,E1 -1011.503,E2 -1011.503} C_VEL
LIN {X 0,Y 594.39,Z 281.446,A -85,B 0,C 180,E1 -1014.445,E2 -1014.445} C_VEL
LIN {X 0,Y 594.342,Z 281.444,A -85,B 0,C 180,E1 -1017.517,E2 -1017.517} C_VEL
LIN {X 0,Y 594.36,Z 281.451,A -85,B 0,C 180,E1 -1020.56,E2 -1020.56} C_VEL
LIN {X 0,Y 594.367,Z 281.445,A -85,B 0,C 180,E1 -1022.95,E2 -1022.95} C_VEL
LIN {X 0,Y 594.311,Z 281.448,A -85,B 0,C 180,E1 -1025.411,E2 -1025.411} C_VEL
LIN {X 0,Y 594.35,Z 281.444,A -85,B 0,C 180,E1 -1027.942,E2 -1027.942} C_VEL
LIN {X 0,Y 594.353,Z 281.453,A -85,B 0,C 180,E1 -1030.819,E2 -1030.819} C_VEL
LIN {X 0,Y 594.334,Z 281.445,A -85,B 0,C 180,E1 -1033.836,E2 -1033.836} C_VEL
LIN {X 0,Y 594.337,Z 281.451,A -85,B 0,C 180,E1 -1036.697,E2 -1036.697} C_VEL
LIN {X 0,Y 594.334,Z 281.449,A -85,B 0,C 180,E1 -1039.43,E2 -1039.43} C_VEL
LIN {X 0,Y 594.342,Z 281.444,A -85,B 0,C 180,E1 -1042.056,E2 -1042.056} C_VEL
LIN {X 0,Y 594.318,Z 281.45,A -85,B 0,C 180,E1 -1044.679,E2 -1044.679} C_VEL
LIN {X 0,Y 594.333,Z 281.453,A -85,B 0,C 180,E1 -1047.094,E2 -1047.094} C_VEL
LIN {X 0,Y 594.335,Z 281.451,A -85,B 0,C 180,E1 -1049.678,E2 -1049.678} C_VEL
LIN {X 0,Y 594.321,Z 281.452,A -85,B 0,C 180,E1 -1051.77,E2 -1051.77} C_VEL
LIN {X 0,Y 594.33,Z 281.448,A -85,B 0,C 180,E1 -1054.053,E2 -1054.053} C_VEL
LIN {X 0,Y 594.333,Z 281.446,A -85,B 0,C 180,E1 -1056.293,E2 -1056.293} C_VEL
LIN {X 0,Y 594.354,Z 281.446,A -85,B 0,C 180,E1 -1059.222,E2 -1059.222} C_VEL
LIN {X 0,Y 594.308,Z 281.454,A -85,B 0,C 180,E1 -1062.093,E2 -1062.093} C_VEL
LIN {X 0,Y 594.323,Z 281.451,A -85,B 0,C 180,E1 -1064.218,E2 -1064.218} C_VEL
LIN {X 0,Y 594.349,Z 281.447,A -85,B 0,C 180,E1 -1066.32,E2 -1066.32} C_VEL
LIN {X 0,Y 594.32,Z 281.447,A -85,B 0,C 180,E1 -1068.956,E2 -1068.956} C_VEL
LIN {X 0,Y 594.364,Z 281.448,A -85,B 0,C 180,E1 -1071.842,E2 -1071.842} C_VEL
LIN {X 0,Y 594.359,Z 281.446,A -85,B 0,C 180,E1 -1074.572,E2 -1074.572} C_VEL
LIN {X 0,Y 594.354,Z 281.442,A -85,B 0,C 180,E1 -1077.289,E2 -1077.289} C_VEL
LIN {X 0,Y 594.384,Z 281.444,A -85,B 0,C 180,E1 -1080,E2 -1080} C_VEL
LIN {X 0,Y 594.399,Z 281.443,A -85,B 0,C 180,E1 -1082.711,E2 -1082.711} C_VEL
LIN {X 0,Y 594.345,Z 281.444,A -85,B 0,C 180,E1 -1085.428,E2 -1085.428} C_VEL
LIN {X 0,Y 594.331,Z 281.445,A -85,B 0,C 180,E1 -1087.474,E2 -1087.474} C_VEL
LIN {X 0,Y 594.326,Z 281.446,A -85,B 0,C 180,E1 -1089.529,E2 -1089.529} C_VEL
LIN {X 0,Y 594.36,Z 281.442,A -85,B 0,C 180,E1 -1091.596,E2 -1091.596} C_VEL
LIN {X 0,Y 594.37,Z 281.445,A -85,B 0,C 180,E1 -1094.377,E2 -1094.377} C_VEL
LIN {X 0,Y 594.364,Z 281.447,A -85,B 0,C 180,E1 -1097.194,E2 -1097.194} C_VEL
LIN {X 0,Y 594.346,Z 281.444,A -85,B 0,C 180,E1 -1100.055,E2 -1100.055} C_VEL
LIN {X 0,Y 594.341,Z 281.454,A -85,B 0,C 180,E1 -1102.968,E2 -1102.968} C_VEL
LIN {X 0,Y 594.353,Z 281.443,A -85,B 0,C 180,E1 -1105.945,E2 -1105.945} C_VEL
LIN {X 0,Y 594.346,Z 281.444,A -85,B 0,C 180,E1 -1108.229,E2 -1108.229} C_VEL
LIN {X 0,Y 594.358,Z 281.443,A -85,B 0,C 180,E1 -1110.561,E2 -1110.561} C_VEL
LIN {X 0,Y 594.366,Z 281.445,A -85,B 0,C 180,E1 -1112.951,E2 -1112.951} C_VEL
LIN {X 0,Y 594.339,Z 281.455,A -85,B 0,C 180,E1 -1115.41,E2 -1115.41} C_VEL
LIN {X 0,Y 594.374,Z 281.444,A -85,B 0,C 180,E1 -1117.942,E2 -1117.942} C_VEL
LIN {X 0,Y 594.358,Z 281.442,A -85,B 0,C 180,E1 -1120.821,E2 -1120.821} C_VEL
LIN {X 0,Y 594.352,Z 281.447,A -85,B 0,C 180,E1 -1123.301,E2 -1123.301} C_VEL
LIN {X 0,Y 594.355,Z 281.447,A -85,B 0,C 180,E1 -1126.162,E2 -1126.162} C_VEL
LIN {X 0,Y 594.372,Z 281.442,A -85,B 0,C 180,E1 -1128.537,E2 -1128.537} C_VEL
LIN {X 0,Y 594.364,Z 281.443,A -85,B 0,C 180,E1 -1131.298,E2 -1131.298} C_VEL
LIN {X 0,Y 594.344,Z 281.45,A -85,B 0,C 180,E1 -1133.756,E2 -1133.756} C_VEL
LIN {X 0,Y 594.375,Z 281.449,A -85,B 0,C 180,E1 -1136.24,E2 -1136.24} C_VEL
LIN {X 0,Y 594.385,Z 281.442,A -85,B 0,C 180,E1 -1138.652,E2 -1138.652} C_VEL
LIN {X 0,Y 594.373,Z 281.441,A -85,B 0,C 180,E1 -1141.044,E2 -1141.044} C_VEL
LIN {X 0,Y 594.382,Z 281.44,A -85,B 0,C 180,E1 -1143.301,E2 -1143.301} C_VEL
LIN {X 0,Y 594.348,Z 281.445,A -85,B 0,C 180,E1 -1145.575,E2 -1145.575} C_VEL
LIN {X 0,Y 594.391,Z 281.53,A -85,B 0,C 180,E1 -1147.411,E2 -1147.411} C_VEL
LIN {X 0,Y 594.736,Z 287.767,A -85,B 0,C 180,E1 -1148.329,E2 -1148.329} C_VEL
LIN {X 0,Y 594.6,Z 307.305,A -85,B 0,C 180,E1 -1151.125,E2 -1151.125} C_VEL
LIN {X 0,Y 594.513,Z 325.546,A -85,B 0,C 180,E1 -1153.695,E2 -1153.695} C_VEL
LIN {X 0,Y 594.426,Z 345.695,A -85,B 0,C 180,E1 -1156.497,E2 -1156.497} C_VEL
LIN {X 0,Y 594.46,Z 347.195,A -85,B 0,C 180,E1 -1156.672,E2 -1156.672} C_VEL
LIN {X 0,Y 594.743,Z 354.35,A -85,B 0,C 180,E1 -1156.765,E2 -1156.765} C_VEL
LIN {X 0,Y 594.662,Z 454.98,A -85,B 0,C 180,E1 -1157.999,E2 -1157.999} C_VEL
LIN {X 0,Y 594.633,Z 468.24,A -85,B 0,C 180,E1 -1158.302,E2 -1158.302} C_VEL
LIN {X 0,Y 594.565,Z 480.428,A -85,B 0,C 180,E1 -1158.712,E2 -1158.712} C_VEL
LIN {X 0,Y 594.535,Z 492.643,A -85,B 0,C 180,E1 -1159.271,E2 -1159.271} C_VEL
LIN {X 0,Y 594.461,Z 504.209,A -85,B 0,C 180,E1 -1159.958,E2 -1159.958} C_VEL
LIN {X 0,Y 594.412,Z 514.53,A -85,B 0,C 180,E1 -1160.73,E2 -1160.73} C_VEL
LIN {X 0,Y 594.349,Z 523.035,A -85,B 0,C 180,E1 -1161.501,E2 -1161.501} C_VEL
LIN {X 0,Y 594.347,Z 530.965,A -85,B 0,C 180,E1 -1162.356,E2 -1162.356} C_VEL
LIN {X 0,Y 594.28,Z 538.829,A -85,B 0,C 180,E1 -1163.411,E2 -1163.411} C_VEL
LIN {X 0,Y 594.289,Z 545.683,A -85,B 0,C 180,E1 -1164.572,E2 -1164.572} C_VEL
LIN {X 0,Y 594.27,Z 550.374,A -85,B 0,C 180,E1 -1165.592,E2 -1165.592} C_VEL
LIN {X 0,Y 594.268,Z 553.958,A -85,B 0,C 180,E1 -1166.611,E2 -1166.611} C_VEL
LIN {X 0,Y 594.226,Z 555.81,A -85,B 0,C 180,E1 -1167.289,E2 -1167.289} C_VEL
LIN {X 0,Y 594.239,Z 557.202,A -85,B 0,C 180,E1 -1167.967,E2 -1167.967} C_VEL
LIN {X 0,Y 594.239,Z 558.784,A -85,B 0,C 180,E1 -1169.323,E2 -1169.323} C_VEL
LIN {X 0,Y 594.236,Z 559,A -85,B 0,C 180,E1 -1170,E2 -1170} C_VEL
LIN {X 0,Y 594.247,Z 558.184,A -85,B 0,C 180,E1 -1171.356,E2 -1171.356} C_VEL
LIN {X 0,Y 594.239,Z 557.201,A -85,B 0,C 180,E1 -1172.034,E2 -1172.034} C_VEL
LIN {X 0,Y 594.226,Z 555.808,A -85,B 0,C 180,E1 -1172.712,E2 -1172.712} C_VEL
LIN {X 0,Y 594.288,Z 552.895,A -85,B 0,C 180,E1 -1173.73,E2 -1173.73} C_VEL
LIN {X 0,Y 594.241,Z 548.948,A -85,B 0,C 180,E1 -1174.749,E2 -1174.749} C_VEL
LIN {X 0,Y 594.304,Z 542.875,A -85,B 0,C 180,E1 -1175.94,E2 -1175.94} C_VEL
LIN {X 0,Y 594.308,Z 536.233,A -85,B 0,C 180,E1 -1176.962,E2 -1176.962} C_VEL
LIN {X 0,Y 594.359,Z 527.986,A -85,B 0,C 180,E1 -1177.987,E2 -1177.987} C_VEL
LIN {X 0,Y 594.383,Z 519.533,A -85,B 0,C 180,E1 -1178.843,E2 -1178.843} C_VEL
LIN {X 0,Y 594.42,Z 509.089,A -85,B 0,C 180,E1 -1179.7,E2 -1179.7} C_VEL
LIN {X 0,Y 594.485,Z 498.752,A -85,B 0,C 180,E1 -1180.387,E2 -1180.387} C_VEL
LIN {X 0,Y 594.56,Z 487.696,A -85,B 0,C 180,E1 -1180.974,E2 -1180.974} C_VEL
LIN {X 0,Y 594.59,Z 475.693,A -85,B 0,C 180,E1 -1181.465,E2 -1181.465} C_VEL
LIN {X 0,Y 594.646,Z 462.334,A -85,B 0,C 180,E1 -1181.85,E2 -1181.85} C_VEL
LIN {X 0,Y 594.693,Z 449.055,A -85,B 0,C 180,E1 -1182.087,E2 -1182.087} C_VEL
LIN {X 0,Y 594.703,Z 348.9,A -85,B 0,C 180,E1 -1183.302,E2 -1183.302} C_VEL
LIN {X 0,Y 594.422,Z 346.79,A -85,B 0,C 180,E1 -1183.352,E2 -1183.352} C_VEL
LIN {X 0,Y 594.51,Z 326.798,A -85,B 0,C 180,E1 -1186.13,E2 -1186.13} C_VEL
LIN {X 0,Y 594.555,Z 309.168,A -85,B 0,C 180,E1 -1188.612,E2 -1188.612} C_VEL
LIN {X 0,Y 594.712,Z 290.078,A -85,B 0,C 180,E1 -1191.338,E2 -1191.338} C_VEL
LIN {X 0,Y 594.465,Z 282.024,A -85,B 0,C 180,E1 -1192.514,E2 -1192.514} C_VEL
LIN {X 0,Y 594.38,Z 281.445,A -85,B 0,C 180,E1 -1192.622,E2 -1192.622} C_VEL
LIN {X 0,Y 594.377,Z 281.445,A -85,B 0,C 180,E1 -1195.193,E2 -1195.193} C_VEL
LIN {X 0,Y 594.39,Z 281.447,A -85,B 0,C 180,E1 -1197.527,E2 -1197.527} C_VEL
LIN {X 0,Y 594.371,Z 281.444,A -85,B 0,C 180,E1 -1200.325,E2 -1200.325} C_VEL
LIN {X 0,Y 594.377,Z 281.44,A -85,B 0,C 180,E1 -1202.95,E2 -1202.95} C_VEL
LIN {X 0,Y 594.348,Z 281.446,A -85,B 0,C 180,E1 -1205.409,E2 -1205.409} C_VEL
LIN {X 0,Y 594.385,Z 281.447,A -85,B 0,C 180,E1 -1207.941,E2 -1207.941} C_VEL
LIN {X 0,Y 594.367,Z 281.443,A -85,B 0,C 180,E1 -1210.821,E2 -1210.821} C_VEL
LIN {X 0,Y 594.352,Z 281.443,A -85,B 0,C 180,E1 -1213.301,E2 -1213.301} C_VEL
LIN {X 0,Y 594.361,Z 281.448,A -85,B 0,C 180,E1 -1216.161,E2 -1216.161} C_VEL
LIN {X 0,Y 594.38,Z 281.451,A -85,B 0,C 180,E1 -1218.536,E2 -1218.536} C_VEL
LIN {X 0,Y 594.369,Z 281.442,A -85,B 0,C 180,E1 -1221.298,E2 -1221.298} C_VEL
LIN {X 0,Y 594.348,Z 281.443,A -85,B 0,C 180,E1 -1223.755,E2 -1223.755} C_VEL
LIN {X 0,Y 594.376,Z 281.442,A -85,B 0,C 180,E1 -1226.239,E2 -1226.239} C_VEL
LIN {X 0,Y 594.376,Z 281.446,A -85,B 0,C 180,E1 -1228.65,E2 -1228.65} C_VEL
LIN {X 0,Y 594.379,Z 281.45,A -85,B 0,C 180,E1 -1231.043,E2 -1231.043} C_VEL
LIN {X 0,Y 594.38,Z 281.447,A -85,B 0,C 180,E1 -1233.3,E2 -1233.3} C_VEL
LIN {X 0,Y 594.345,Z 281.448,A -85,B 0,C 180,E1 -1235.575,E2 -1235.575} C_VEL
LIN {X 0,Y 594.358,Z 281.443,A -85,B 0,C 180,E1 -1238.496,E2 -1238.496} C_VEL
LIN {X 0,Y 594.375,Z 281.452,A -85,B 0,C 180,E1 -1241.382,E2 -1241.382} C_VEL
LIN {X 0,Y 594.403,Z 281.447,A -85,B 0,C 180,E1 -1243.515,E2 -1243.515} C_VEL
LIN {X 0,Y 594.363,Z 281.442,A -85,B 0,C 180,E1 -1246.321,E2 -1246.321} C_VEL
LIN {X 0,Y 594.38,Z 281.441,A -85,B 0,C 180,E1 -1249.095,E2 -1249.095} C_VEL
LIN {X 0,Y 594.378,Z 281.45,A -85,B 0,C 180,E1 -1251.843,E2 -1251.843} C_VEL
LIN {X 0,Y 594.369,Z 281.441,A -85,B 0,C 180,E1 -1254.572,E2 -1254.572} C_VEL
LIN {X 0,Y 594.405,Z 281.437,A -85,B 0,C 180,E1 -1257.289,E2 -1257.289} C_VEL
LIN {X 0,Y 594.417,Z 281.445,A -85,B 0,C 180,E1 -1260,E2 -1260} C_VEL
LIN {X 0,Y 594.387,Z 281.441,A -85,B 0,C 180,E1 -1262.711,E2 -1262.711} C_VEL
LIN {X 0,Y 594.379,Z 281.439,A -85,B 0,C 180,E1 -1265.428,E2 -1265.428} C_VEL
LIN {X 0,Y 594.412,Z 281.442,A -85,B 0,C 180,E1 -1268.157,E2 -1268.157} C_VEL
LIN {X 0,Y 594.373,Z 281.442,A -85,B 0,C 180,E1 -1271.066,E2 -1271.066} C_VEL
LIN {X 0,Y 594.37,Z 281.44,A -85,B 0,C 180,E1 -1273.679,E2 -1273.679} C_VEL
LIN {X 0,Y 594.35,Z 281.445,A -85,B 0,C 180,E1 -1275.315,E2 -1275.315} C_VEL
LIN {X 0,Y 593.672,Z 281.53,A -85,B 0,C 180,E1 -1275.881,E2 -1275.881} C_VEL
LIN {X 0,Y 590.8,Z 281.895,A -85,B 0,C 180,E1 -1276.799,E2 -1276.799} C_VEL
LIN {X 0,Y 588.391,Z 282.19,A -85,B 0,C 180,E1 -1277.538,E2 -1277.538} C_VEL
LIN {X 0,Y 587.372,Z 282.313,A -85,B 0,C 180,E1 -1278.108,E2 -1278.108} C_VEL
LIN {X 0,Y 587.298,Z 282.324,A -85,B 0,C 180,E1 -1278.301,E2 -1278.301} C_VEL
LIN {X 0,Y 587.332,Z 282.325,A -85,B 0,C 180,E1 -1281.038,E2 -1281.038} C_VEL
LIN {X 0,Y 587.308,Z 282.326,A -85,B 0,C 180,E1 -1283.26,E2 -1283.26} C_VEL
LIN {X 0,Y 587.319,Z 282.322,A -85,B 0,C 180,E1 -1285.518,E2 -1285.518} C_VEL
LIN {X 0,Y 587.306,Z 282.321,A -85,B 0,C 180,E1 -1287.82,E2 -1287.82} C_VEL
LIN {X 0,Y 587.321,Z 282.319,A -85,B 0,C 180,E1 -1290.507,E2 -1290.507} C_VEL
LIN {X 0,Y 587.337,Z 282.324,A -85,B 0,C 180,E1 -1293.111,E2 -1293.111} C_VEL
LIN {X 0,Y 587.301,Z 282.331,A -85,B 0,C 180,E1 -1295.538,E2 -1295.538} C_VEL
LIN {X 0,Y 587.321,Z 282.319,A -85,B 0,C 180,E1 -1298.48,E2 -1298.48} C_VEL
LIN {X 0,Y 587.336,Z 282.32,A -85,B 0,C 180,E1 -1301.157,E2 -1301.157} C_VEL
LIN {X 0,Y 587.316,Z 282.325,A -85,B 0,C 180,E1 -1304.112,E2 -1304.112} C_VEL
LIN {X 0,Y 587.306,Z 282.321,A -85,B 0,C 180,E1 -1306.993,E2 -1306.993} C_VEL
LIN {X 0,Y 587.311,Z 282.327,A -85,B 0,C 180,E1 -1309.745,E2 -1309.745} C_VEL
LIN {X 0,Y 587.322,Z 282.325,A -85,B 0,C 180,E1 -1312.39,E2 -1312.39} C_VEL
LIN {X 0,Y 587.337,Z 282.32,A -85,B 0,C 180,E1 -1315.655,E2 -1315.655} C_VEL
LIN {X 0,Y 587.341,Z 282.328,A -85,B 0,C 180,E1 -1318.231,E2 -1318.231} C_VEL
LIN {X 0,Y 587.36,Z 282.389,A -85,B 0,C 180,E1 -1319.457,E2 -1319.457} C_VEL
LIN {X 0,Y 587.455,Z 290.432,A -85,B 0,C 180,E1 -1320.849,E2 -1320.849} C_VEL
LIN {X 0,Y 587.41,Z 305.026,A -85,B 0,C 180,E1 -1323.342,E2 -1323.342} C_VEL
LIN {X 0,Y 587.381,Z 318.161,A -85,B 0,C 180,E1 -1325.56,E2 -1325.56} C_VEL
LIN {X 0,Y 587.887,Z 323.641,A -85,B 0,C 180,E1 -1325.644,E2 -1325.644} C_VEL
LIN {X 0,Y 587.727,Z 425.257,A -85,B 0,C 180,E1 -1326.906,E2 -1326.906} C_VEL
LIN {X 0,Y 587.651,Z 438.702,A -85,B 0,C 180,E1 -1327.219,E2 -1327.219} C_VEL
LIN {X 0,Y 587.609,Z 451.942,A -85,B 0,C 180,E1 -1327.682,E2 -1327.682} C_VEL
LIN {X 0,Y 587.515,Z 463.495,A -85,B 0,C 180,E1 -1328.233,E2 -1328.233} C_VEL
LIN {X 0,Y 587.458,Z 475.458,A -85,B 0,C 180,E1 -1328.967,E2 -1328.967} C_VEL
LIN {X 0,Y 587.375,Z 484.937,A -85,B 0,C 180,E1 -1329.697,E2 -1329.697} C_VEL
LIN {X 0,Y 587.366,Z 492.87,A -85,B 0,C 180,E1 -1330.425,E2 -1330.425} C_VEL
LIN {X 0,Y 587.265,Z 501.138,A -85,B 0,C 180,E1 -1331.329,E2 -1331.329} C_VEL
LIN {X 0,Y 587.222,Z 509.049,A -85,B 0,C 180,E1 -1332.41,E2 -1332.41} C_VEL
LIN {X 0,Y 587.188,Z 514.395,A -85,B 0,C 180,E1 -1333.306,E2 -1333.306} C_VEL
LIN {X 0,Y 587.186,Z 519.52,A -85,B 0,C 180,E1 -1334.377,E2 -1334.377} C_VEL
LIN {X 0,Y 587.149,Z 523.427,A -85,B 0,C 180,E1 -1335.441,E2 -1335.441} C_VEL
LIN {X 0,Y 587.187,Z 525.423,A -85,B 0,C 180,E1 -1336.15,E2 -1336.15} C_VEL
LIN {X 0,Y 587.146,Z 526.975,A -85,B 0,C 180,E1 -1336.854,E2 -1336.854} C_VEL
LIN {X 0,Y 587.161,Z 528.053,A -85,B 0,C 180,E1 -1337.558,E2 -1337.558} C_VEL
LIN {X 0,Y 587.169,Z 528.987,A -85,B 0,C 180,E1 -1338.959,E2 -1338.959} C_VEL
LIN {X 0,Y 587.142,Z 528.835,A -85,B 0,C 180,E1 -1339.656,E2 -1339.656} C_VEL
LIN {X 0,Y 587.152,Z 528.258,A -85,B 0,C 180,E1 -1340.353,E2 -1340.353} C_VEL
LIN {X 0,Y 587.129,Z 527.291,A -85,B 0,C 180,E1 -1341.047,E2 -1341.047} C_VEL
LIN {X 0,Y 587.14,Z 525.92,A -85,B 0,C 180,E1 -1341.741,E2 -1341.741} C_VEL
LIN {X 0,Y 587.158,Z 523.021,A -85,B 0,C 180,E1 -1342.78,E2 -1342.78} C_VEL
LIN {X 0,Y 587.18,Z 519.097,A -85,B 0,C 180,E1 -1343.816,E2 -1343.816} C_VEL
LIN {X 0,Y 587.188,Z 514.05,A -85,B 0,C 180,E1 -1344.849,E2 -1344.849} C_VEL
LIN {X 0,Y 587.23,Z 507.729,A -85,B 0,C 180,E1 -1345.882,E2 -1345.882} C_VEL
LIN {X 0,Y 587.27,Z 499.846,A -85,B 0,C 180,E1 -1346.913,E2 -1346.913} C_VEL
LIN {X 0,Y 587.355,Z 490.083,A -85,B 0,C 180,E1 -1347.942,E2 -1347.942} C_VEL
LIN {X 0,Y 587.38,Z 479.927,A -85,B 0,C 180,E1 -1348.8,E2 -1348.8} C_VEL
LIN {X 0,Y 587.458,Z 468.526,A -85,B 0,C 180,E1 -1349.571,E2 -1349.571} C_VEL
LIN {X 0,Y 587.571,Z 457.302,A -85,B 0,C 180,E1 -1350.171,E2 -1350.171} C_VEL
LIN {X 0,Y 587.608,Z 444.599,A -85,B 0,C 180,E1 -1350.685,E2 -1350.685} C_VEL
LIN {X 0,Y 587.678,Z 431.889,A -85,B 0,C 180,E1 -1351.049,E2 -1351.049} C_VEL
LIN {X 0,Y 587.753,Z 418.51,A -85,B 0,C 180,E1 -1351.284,E2 -1351.284} C_VEL
LIN {X 0,Y 587.769,Z 320.77,A -85,B 0,C 180,E1 -1352.484,E2 -1352.484} C_VEL
LIN {X 0,Y 587.372,Z 318.174,A -85,B 0,C 180,E1 -1352.528,E2 -1352.528} C_VEL
LIN {X 0,Y 587.42,Z 302.675,A -85,B 0,C 180,E1 -1355.148,E2 -1355.148} C_VEL
LIN {X 0,Y 587.55,Z 286.555,A -85,B 0,C 180,E1 -1357.906,E2 -1357.906} C_VEL
LIN {X 0,Y 587.293,Z 282.328,A -85,B 0,C 180,E1 -1358.667,E2 -1358.667} C_VEL
LIN {X 0,Y 587.335,Z 282.319,A -85,B 0,C 180,E1 -1361.124,E2 -1361.124} C_VEL
LIN {X 0,Y 587.331,Z 282.323,A -85,B 0,C 180,E1 -1364.245,E2 -1364.245} C_VEL
LIN {X 0,Y 587.283,Z 282.324,A -85,B 0,C 180,E1 -1366.791,E2 -1366.791} C_VEL
LIN {X 0,Y 587.302,Z 282.324,A -85,B 0,C 180,E1 -1369.576,E2 -1369.576} C_VEL
LIN {X 0,Y 587.305,Z 282.325,A -85,B 0,C 180,E1 -1371.774,E2 -1371.774} C_VEL
LIN {X 0,Y 587.307,Z 282.323,A -85,B 0,C 180,E1 -1374.76,E2 -1374.76} C_VEL
LIN {X 0,Y 587.299,Z 282.323,A -85,B 0,C 180,E1 -1377.682,E2 -1377.682} C_VEL
LIN {X 0,Y 587.316,Z 282.329,A -85,B 0,C 180,E1 -1380.506,E2 -1380.506} C_VEL
LIN {X 0,Y 587.313,Z 282.32,A -85,B 0,C 180,E1 -1383.397,E2 -1383.397} C_VEL
LIN {X 0,Y 587.272,Z 282.326,A -85,B 0,C 180,E1 -1385.9,E2 -1385.9} C_VEL
LIN {X 0,Y 587.304,Z 282.328,A -85,B 0,C 180,E1 -1388.48,E2 -1388.48} C_VEL
LIN {X 0,Y 587.29,Z 282.327,A -85,B 0,C 180,E1 -1391.16,E2 -1391.16} C_VEL
LIN {X 0,Y 587.296,Z 282.322,A -85,B 0,C 180,E1 -1394.11,E2 -1394.11} C_VEL
LIN {X 0,Y 587.279,Z 282.335,A -85,B 0,C 180,E1 -1396.99,E2 -1396.99} C_VEL
LIN {X 0,Y 587.284,Z 282.324,A -85,B 0,C 180,E1 -1399.743,E2 -1399.743} C_VEL
LIN {X 0,Y 587.301,Z 282.322,A -85,B 0,C 180,E1 -1402.389,E2 -1402.389} C_VEL
LIN {X 0,Y 587.322,Z 282.323,A -85,B 0,C 180,E1 -1405.654,E2 -1405.654} C_VEL
LIN {X 0,Y 587.29,Z 282.323,A -85,B 0,C 180,E1 -1408.228,E2 -1408.228} C_VEL
LIN {X 0,Y 587.312,Z 282.322,A -85,B 0,C 180,E1 -1410.871,E2 -1410.871} C_VEL
LIN {X 0,Y 587.284,Z 282.329,A -85,B 0,C 180,E1 -1413.832,E2 -1413.832} C_VEL
LIN {X 0,Y 587.286,Z 282.323,A -85,B 0,C 180,E1 -1416.739,E2 -1416.739} C_VEL
LIN {X 0,Y 587.291,Z 282.334,A -85,B 0,C 180,E1 -1419.694,E2 -1419.694} C_VEL
LIN {X 0,Y 587.264,Z 282.335,A -85,B 0,C 180,E1 -1421.871,E2 -1421.871} C_VEL
LIN {X 0,Y 587.265,Z 282.326,A -85,B 0,C 180,E1 -1424.735,E2 -1424.735} C_VEL
LIN {X 0,Y 587.258,Z 282.327,A -85,B 0,C 180,E1 -1426.857,E2 -1426.857} C_VEL
LIN {X 0,Y 587.31,Z 282.325,A -85,B 0,C 180,E1 -1429.659,E2 -1429.659} C_VEL
LIN {X 0,Y 587.301,Z 282.326,A -85,B 0,C 180,E1 -1432.436,E2 -1432.436} C_VEL
LIN {X 0,Y 587.309,Z 282.32,A -85,B 0,C 180,E1 -1435.195,E2 -1435.195} C_VEL
LIN {X 0,Y 587.341,Z 282.322,A -85,B 0,C 180,E1 -1437.943,E2 -1437.943} C_VEL
LIN {X 0,Y 587.378,Z 282.317,A -85,B 0,C 180,E1 -1440.685,E2 -1440.685} C_VEL
LIN {X 0,Y 587.361,Z 282.319,A -85,B 0,C 180,E1 -1442.743,E2 -1442.743} C_VEL
LIN {X 0,Y 587.313,Z 282.32,A -85,B 0,C 180,E1 -1445.493,E2 -1445.493} C_VEL
LIN {X 0,Y 587.293,Z 282.322,A -85,B 0,C 180,E1 -1447.564,E2 -1447.564} C_VEL
LIN {X 0,Y 587.292,Z 282.328,A -85,B 0,C 180,E1 -1450.341,E2 -1450.341} C_VEL
LIN {X 0,Y 587.293,Z 282.327,A -85,B 0,C 180,E1 -1453.142,E2 -1453.142} C_VEL
LIN {X 0,Y 587.31,Z 282.324,A -85,B 0,C 180,E1 -1455.264,E2 -1455.264} C_VEL
LIN {X 0,Y 587.296,Z 282.324,A -85,B 0,C 180,E1 -1457.408,E2 -1457.408} C_VEL
LIN {X 0,Y 587.294,Z 282.324,A -85,B 0,C 180,E1 -1459.577,E2 -1459.577} C_VEL
LIN {X 0,Y 587.3,Z 282.322,A -85,B 0,C 180,E1 -1461.775,E2 -1461.775} C_VEL
LIN {X 0,Y 587.295,Z 282.327,A -85,B 0,C 180,E1 -1464.761,E2 -1464.761} C_VEL
LIN {X 0,Y 587.326,Z 282.32,A -85,B 0,C 180,E1 -1467.819,E2 -1467.819} C_VEL
LIN {X 0,Y 587.312,Z 282.32,A -85,B 0,C 180,E1 -1470.508,E2 -1470.508} C_VEL
LIN {X 0,Y 587.329,Z 282.324,A -85,B 0,C 180,E1 -1473.112,E2 -1473.112} C_VEL
LIN {X 0,Y 587.287,Z 282.333,A -85,B 0,C 180,E1 -1475.538,E2 -1475.538} C_VEL
LIN {X 0,Y 587.311,Z 282.32,A -85,B 0,C 180,E1 -1478.481,E2 -1478.481} C_VEL
LIN {X 0,Y 587.325,Z 282.321,A -85,B 0,C 180,E1 -1481.158,E2 -1481.158} C_VEL
LIN {X 0,Y 587.306,Z 282.325,A -85,B 0,C 180,E1 -1484.113,E2 -1484.113} C_VEL
LIN {X 0,Y 587.29,Z 282.323,A -85,B 0,C 180,E1 -1486.993,E2 -1486.993} C_VEL
LIN {X 0,Y 587.304,Z 282.329,A -85,B 0,C 180,E1 -1489.746,E2 -1489.746} C_VEL
LIN {X 0,Y 587.338,Z 282.321,A -85,B 0,C 180,E1 -1492.393,E2 -1492.393} C_VEL
LIN {X 0,Y 587.35,Z 282.32,A -85,B 0,C 180,E1 -1495.78,E2 -1495.78} C_VEL
LIN {X 0,Y 587.344,Z 282.327,A -85,B 0,C 180,E1 -1498.232,E2 -1498.232} C_VEL
LIN {X 0,Y 587.342,Z 282.318,A -85,B 0,C 180,E1 -1500.868,E2 -1500.868} C_VEL
LIN {X 0,Y 587.329,Z 282.32,A -85,B 0,C 180,E1 -1503.722,E2 -1503.722} C_VEL
LIN {X 0,Y 587.304,Z 282.326,A -85,B 0,C 180,E1 -1505.993,E2 -1505.993} C_VEL
LIN {X 0,Y 587.343,Z 282.449,A -85,B 0,C 180,E1 -1507.26,E2 -1507.26} C_VEL
LIN {X 0,Y 587.801,Z 286.507,A -85,B 0,C 180,E1 -1507.876,E2 -1507.876} C_VEL
LIN {X 0,Y 587.664,Z 306.069,A -85,B 0,C 180,E1 -1510.715,E2 -1510.715} C_VEL
LIN {X 0,Y 587.534,Z 325.546,A -85,B 0,C 180,E1 -1513.496,E2 -1513.496} C_VEL
LIN {X 0,Y 587.404,Z 346.325,A -85,B 0,C 180,E1 -1516.421,E2 -1516.421} C_VEL
LIN {X 0,Y 587.426,Z 347.195,A -85,B 0,C 180,E1 -1516.509,E2 -1516.509} C_VEL
LIN {X 0,Y 587.879,Z 352.561,A -85,B 0,C 180,E1 -1516.586,E2 -1516.586} C_VEL
LIN {X 0,Y 587.724,Z 454.98,A -85,B 0,C 180,E1 -1517.856,E2 -1517.856} C_VEL
LIN {X 0,Y 587.679,Z 468.241,A -85,B 0,C 180,E1 -1518.161,E2 -1518.161} C_VEL
LIN {X 0,Y 587.592,Z 480.617,A -85,B 0,C 180,E1 -1518.584,E2 -1518.584} C_VEL
LIN {X 0,Y 587.552,Z 492.642,A -85,B 0,C 180,E1 -1519.142,E2 -1519.142} C_VEL
LIN {X 0,Y 587.457,Z 504.211,A -85,B 0,C 180,E1 -1519.837,E2 -1519.837} C_VEL
LIN {X 0,Y 587.362,Z 514.546,A -85,B 0,C 180,E1 -1520.618,E2 -1520.618} C_VEL
LIN {X 0,Y 587.298,Z 523.048,A -85,B 0,C 180,E1 -1521.398,E2 -1521.398} C_VEL
LIN {X 0,Y 587.273,Z 530.965,A -85,B 0,C 180,E1 -1522.263,E2 -1522.263} C_VEL
LIN {X 0,Y 587.229,Z 537.473,A -85,B 0,C 180,E1 -1523.127,E2 -1523.127} C_VEL
LIN {X 0,Y 587.236,Z 543.87,A -85,B 0,C 180,E1 -1524.162,E2 -1524.162} C_VEL
LIN {X 0,Y 587.147,Z 548.952,A -85,B 0,C 180,E1 -1525.194,E2 -1525.194} C_VEL
LIN {X 0,Y 587.212,Z 552.897,A -85,B 0,C 180,E1 -1526.226,E2 -1526.226} C_VEL
LIN {X 0,Y 587.132,Z 555.81,A -85,B 0,C 180,E1 -1527.256,E2 -1527.256} C_VEL
LIN {X 0,Y 587.138,Z 557.201,A -85,B 0,C 180,E1 -1527.943,E2 -1527.943} C_VEL
LIN {X 0,Y 587.14,Z 558.785,A -85,B 0,C 180,E1 -1529.315,E2 -1529.315} C_VEL
LIN {X 0,Y 587.137,Z 559,A -85,B 0,C 180,E1 -1530.001,E2 -1530.001} C_VEL
LIN {X 0,Y 587.147,Z 558.185,A -85,B 0,C 180,E1 -1531.372,E2 -1531.372} C_VEL
LIN {X 0,Y 587.138,Z 557.2,A -85,B 0,C 180,E1 -1532.058,E2 -1532.058} C_VEL
LIN {X 0,Y 587.132,Z 555.809,A -85,B 0,C 180,E1 -1532.745,E2 -1532.745} C_VEL
LIN {X 0,Y 587.212,Z 552.894,A -85,B 0,C 180,E1 -1533.775,E2 -1533.775} C_VEL
LIN {X 0,Y 587.147,Z 548.947,A -85,B 0,C 180,E1 -1534.807,E2 -1534.807} C_VEL
LIN {X 0,Y 587.217,Z 542.875,A -85,B 0,C 180,E1 -1536.012,E2 -1536.012} C_VEL
LIN {X 0,Y 587.245,Z 536.234,A -85,B 0,C 180,E1 -1537.047,E2 -1537.047} C_VEL
LIN {X 0,Y 587.297,Z 527.986,A -85,B 0,C 180,E1 -1538.083,E2 -1538.083} C_VEL
LIN {X 0,Y 587.348,Z 519.533,A -85,B 0,C 180,E1 -1538.949,E2 -1538.949} C_VEL
LIN {X 0,Y 587.406,Z 509.09,A -85,B 0,C 180,E1 -1539.817,E2 -1539.817} C_VEL
LIN {X 0,Y 587.501,Z 498.751,A -85,B 0,C 180,E1 -1540.512,E2 -1540.512} C_VEL
LIN {X 0,Y 587.584,Z 486.802,A -85,B 0,C 180,E1 -1541.149,E2 -1541.149} C_VEL
LIN {X 0,Y 587.638,Z 474.584,A -85,B 0,C 180,E1 -1541.64,E2 -1541.64} C_VEL
LIN {X 0,Y 587.684,Z 461.419,A -85,B 0,C 180,E1 -1542.015,E2 -1542.015} C_VEL
LIN {X 0,Y 587.776,Z 449.055,A -85,B 0,C 180,E1 -1542.232,E2 -1542.232} C_VEL
LIN {X 0,Y 587.704,Z 348.902,A -85,B 0,C 180,E1 -1543.463,E2 -1543.463} C_VEL
LIN {X 0,Y 587.381,Z 346.79,A -85,B 0,C 180,E1 -1543.515,E2 -1543.515} C_VEL
LIN {X 0,Y 587.517,Z 328.057,A -85,B 0,C 180,E1 -1546.148,E2 -1546.148} C_VEL
LIN {X 0,Y 587.612,Z 309.168,A -85,B 0,C 180,E1 -1548.84,E2 -1548.84} C_VEL
LIN {X 0,Y 587.776,Z 291.496,A -85,B 0,C 180,E1 -1551.395,E2 -1551.395} C_VEL
LIN {X 0,Y 587.609,Z 283.981,A -85,B 0,C 180,E1 -1552.503,E2 -1552.503} C_VEL
LIN {X 0,Y 587.325,Z 282.326,A -85,B 0,C 180,E1 -1552.79,E2 -1552.79} C_VEL
LIN {X 0,Y 587.334,Z 282.328,A -85,B 0,C 180,E1 -1555.517,E2 -1555.517} C_VEL
LIN {X 0,Y 587.346,Z 282.327,A -85,B 0,C 180,E1 -1557.818,E2 -1557.818} C_VEL
LIN {X 0,Y 587.326,Z 282.321,A -85,B 0,C 180,E1 -1560.508,E2 -1560.508} C_VEL
LIN {X 0,Y 587.339,Z 282.318,A -85,B 0,C 180,E1 -1563.111,E2 -1563.111} C_VEL
LIN {X 0,Y 587.295,Z 282.326,A -85,B 0,C 180,E1 -1565.537,E2 -1565.537} C_VEL
LIN {X 0,Y 587.34,Z 282.323,A -85,B 0,C 180,E1 -1567.838,E2 -1567.838} C_VEL
LIN {X 0,Y 587.309,Z 282.331,A -85,B 0,C 180,E1 -1570.255,E2 -1570.255} C_VEL
LIN {X 0,Y 587.303,Z 282.321,A -85,B 0,C 180,E1 -1573.117,E2 -1573.117} C_VEL
LIN {X 0,Y 587.313,Z 282.325,A -85,B 0,C 180,E1 -1576.048,E2 -1576.048} C_VEL
LIN {X 0,Y 587.334,Z 282.321,A -85,B 0,C 180,E1 -1578.925,E2 -1578.925} C_VEL
LIN {X 0,Y 587.319,Z 282.319,A -85,B 0,C 180,E1 -1581.52,E2 -1581.52} C_VEL
LIN {X 0,Y 587.289,Z 282.324,A -85,B 0,C 180,E1 -1584.1,E2 -1584.1} C_VEL
LIN {X 0,Y 587.333,Z 282.325,A -85,B 0,C 180,E1 -1586.603,E2 -1586.603} C_VEL
LIN {X 0,Y 587.327,Z 282.327,A -85,B 0,C 180,E1 -1589.033,E2 -1589.033} C_VEL
LIN {X 0,Y 587.314,Z 282.324,A -85,B 0,C 180,E1 -1591.402,E2 -1591.402} C_VEL
LIN {X 0,Y 587.308,Z 282.321,A -85,B 0,C 180,E1 -1593.829,E2 -1593.829} C_VEL
LIN {X 0,Y 587.295,Z 282.322,A -85,B 0,C 180,E1 -1595.992,E2 -1595.992} C_VEL
LIN {X 0,Y 587.331,Z 282.323,A -85,B 0,C 180,E1 -1598.962,E2 -1598.962} C_VEL
LIN {X 0,Y 587.349,Z 282.322,A -85,B 0,C 180,E1 -1601.151,E2 -1601.151} C_VEL
LIN {X 0,Y 587.314,Z 282.322,A -85,B 0,C 180,E1 -1604.025,E2 -1604.025} C_VEL
LIN {X 0,Y 587.343,Z 282.317,A -85,B 0,C 180,E1 -1606.154,E2 -1606.154} C_VEL
LIN {X 0,Y 587.345,Z 282.316,A -85,B 0,C 180,E1 -1608.963,E2 -1608.963} C_VEL
LIN {X 0,Y 587.339,Z 282.327,A -85,B 0,C 180,E1 -1611.744,E2 -1611.744} C_VEL
LIN {X 0,Y 587.316,Z 282.33,A -85,B 0,C 180,E1 -1613.818,E2 -1613.818} C_VEL
LIN {X 0,Y 587.314,Z 282.33,A -85,B 0,C 180,E1 -1615.883,E2 -1615.883} C_VEL
LIN {X 0,Y 587.374,Z 282.322,A -85,B 0,C 180,E1 -1617.943,E2 -1617.943} C_VEL
LIN {X 0,Y 587.372,Z 282.314,A -85,B 0,C 180,E1 -1620.686,E2 -1620.686} C_VEL
LIN {X 0,Y 587.317,Z 282.319,A -85,B 0,C 180,E1 -1623.43,E2 -1623.43} C_VEL
LIN {X 0,Y 587.331,Z 282.326,A -85,B 0,C 180,E1 -1626.183,E2 -1626.183} C_VEL
LIN {X 0,Y 587.317,Z 282.321,A -85,B 0,C 180,E1 -1628.95,E2 -1628.95} C_VEL
LIN {X 0,Y 587.326,Z 282.319,A -85,B 0,C 180,E1 -1631.737,E2 -1631.737} C_VEL
LIN {X 0,Y 587.337,Z 282.326,A -85,B 0,C 180,E1 -1634.554,E2 -1634.554} C_VEL
LIN {X 0,Y 587.34,Z 282.317,A -85,B 0,C 180,E1 -1637.407,E2 -1637.407} C_VEL
LIN {X 0,Y 587.298,Z 282.324,A -85,B 0,C 180,E1 -1638.301,E2 -1638.301} C_VEL
LIN {X 0,Y 586.662,Z 282.411,A -85,B 0,C 180,E1 -1638.873,E2 -1638.873} C_VEL
LIN {X 0,Y 583.845,Z 282.764,A -85,B 0,C 180,E1 -1639.802,E2 -1639.802} C_VEL
LIN {X 0,Y 581.436,Z 283.062,A -85,B 0,C 180,E1 -1640.549,E2 -1640.549} C_VEL
LIN {X 0,Y 580.38,Z 283.19,A -85,B 0,C 180,E1 -1641.125,E2 -1641.125} C_VEL
LIN {X 0,Y 580.283,Z 283.199,A -85,B 0,C 180,E1 -1641.32,E2 -1641.32} C_VEL
LIN {X 0,Y 580.264,Z 283.2,A -85,B 0,C 180,E1 -1643.559,E2 -1643.559} C_VEL
LIN {X 0,Y 580.272,Z 283.197,A -85,B 0,C 180,E1 -1645.85,E2 -1645.85} C_VEL
LIN {X 0,Y 580.291,Z 283.201,A -85,B 0,C 180,E1 -1648.977,E2 -1648.977} C_VEL
LIN {X 0,Y 580.301,Z 283.194,A -85,B 0,C 180,E1 -1652.03,E2 -1652.03} C_VEL
LIN {X 0,Y 580.293,Z 283.195,A -85,B 0,C 180,E1 -1654.696,E2 -1654.696} C_VEL
LIN {X 0,Y 580.289,Z 283.202,A -85,B 0,C 180,E1 -1657.27,E2 -1657.27} C_VEL
LIN {X 0,Y 580.291,Z 283.196,A -85,B 0,C 180,E1 -1660.27,E2 -1660.27} C_VEL
LIN {X 0,Y 580.26,Z 283.199,A -85,B 0,C 180,E1 -1662.708,E2 -1662.708} C_VEL
LIN {X 0,Y 580.253,Z 283.207,A -85,B 0,C 180,E1 -1665.611,E2 -1665.611} C_VEL
LIN {X 0,Y 580.26,Z 283.205,A -85,B 0,C 180,E1 -1668.229,E2 -1668.229} C_VEL
LIN {X 0,Y 580.269,Z 283.198,A -85,B 0,C 180,E1 -1670.964,E2 -1670.964} C_VEL
LIN {X 0,Y 580.247,Z 283.204,A -85,B 0,C 180,E1 -1673.595,E2 -1673.595} C_VEL
LIN {X 0,Y 580.299,Z 283.204,A -85,B 0,C 180,E1 -1676.144,E2 -1676.144} C_VEL
LIN {X 0,Y 580.276,Z 283.204,A -85,B 0,C 180,E1 -1678.614,E2 -1678.614} C_VEL
LIN {X 0,Y 580.325,Z 283.302,A -85,B 0,C 180,E1 -1679.37,E2 -1679.37} C_VEL
LIN {X 0,Y 580.517,Z 288.232,A -85,B 0,C 180,E1 -1680.24,E2 -1680.24} C_VEL
LIN {X 0,Y 580.41,Z 303.005,A -85,B 0,C 180,E1 -1682.799,E2 -1682.799} C_VEL
LIN {X 0,Y 580.32,Z 318.108,A -85,B 0,C 180,E1 -1685.383,E2 -1685.383} C_VEL
LIN {X 0,Y 580.97,Z 323.265,A -85,B 0,C 180,E1 -1685.477,E2 -1685.477} C_VEL
LIN {X 0,Y 580.785,Z 425.415,A -85,B 0,C 180,E1 -1686.762,E2 -1686.762} C_VEL
LIN {X 0,Y 580.686,Z 438.895,A -85,B 0,C 180,E1 -1687.081,E2 -1687.081} C_VEL
LIN {X 0,Y 580.642,Z 451.858,A -85,B 0,C 180,E1 -1687.54,E2 -1687.54} C_VEL
LIN {X 0,Y 580.52,Z 464.262,A -85,B 0,C 180,E1 -1688.144,E2 -1688.144} C_VEL
LIN {X 0,Y 580.442,Z 476.084,A -85,B 0,C 180,E1 -1688.887,E2 -1688.887} C_VEL
LIN {X 0,Y 580.345,Z 485.442,A -85,B 0,C 180,E1 -1689.625,E2 -1689.625} C_VEL
LIN {X 0,Y 580.305,Z 493.468,A -85,B 0,C 180,E1 -1690.38,E2 -1690.38} C_VEL
LIN {X 0,Y 580.218,Z 501.471,A -85,B 0,C 180,E1 -1691.277,E2 -1691.277} C_VEL
LIN {X 0,Y 580.137,Z 509.316,A -85,B 0,C 180,E1 -1692.37,E2 -1692.37} C_VEL
LIN {X 0,Y 580.101,Z 515.678,A -85,B 0,C 180,E1 -1693.483,E2 -1693.483} C_VEL
LIN {X 0,Y 580.097,Z 520.425,A -85,B 0,C 180,E1 -1694.541,E2 -1694.541} C_VEL
LIN {X 0,Y 580.089,Z 524.494,A -85,B 0,C 180,E1 -1695.752,E2 -1695.752} C_VEL
LIN {X 0,Y 580.067,Z 526.699,A -85,B 0,C 180,E1 -1696.691,E2 -1696.691} C_VEL
LIN {X 0,Y 580.051,Z 527.892,A -85,B 0,C 180,E1 -1697.403,E2 -1697.403} C_VEL
LIN {X 0,Y 580.055,Z 528.624,A -85,B 0,C 180,E1 -1698.113,E2 -1698.113} C_VEL
LIN {X 0,Y 580.076,Z 528.979,A -85,B 0,C 180,E1 -1698.925,E2 -1698.925} C_VEL
LIN {X 0,Y 580.058,Z 528.41,A -85,B 0,C 180,E1 -1700.234,E2 -1700.234} C_VEL
LIN {X 0,Y 580.062,Z 526.2,A -85,B 0,C 180,E1 -1701.64,E2 -1701.64} C_VEL
LIN {X 0,Y 580.082,Z 523.43,A -85,B 0,C 180,E1 -1702.691,E2 -1702.691} C_VEL
LIN {X 0,Y 580.093,Z 519.645,A -85,B 0,C 180,E1 -1703.74,E2 -1703.74} C_VEL
LIN {X 0,Y 580.102,Z 514.749,A -85,B 0,C 180,E1 -1704.786,E2 -1704.786} C_VEL
LIN {X 0,Y 580.141,Z 508.601,A -85,B 0,C 180,E1 -1705.831,E2 -1705.831} C_VEL
LIN {X 0,Y 580.208,Z 500.978,A -85,B 0,C 180,E1 -1706.875,E2 -1706.875} C_VEL
LIN {X 0,Y 580.304,Z 491.442,A -85,B 0,C 180,E1 -1707.917,E2 -1707.917} C_VEL
LIN {X 0,Y 580.355,Z 480.549,A -85,B 0,C 180,E1 -1708.872,E2 -1708.872} C_VEL
LIN {X 0,Y 580.455,Z 469.282,A -85,B 0,C 180,E1 -1709.653,E2 -1709.653} C_VEL
LIN {X 0,Y 580.584,Z 458.24,A -85,B 0,C 180,E1 -1710.26,E2 -1710.26} C_VEL
LIN {X 0,Y 580.667,Z 445.953,A -85,B 0,C 180,E1 -1710.78,E2 -1710.78} C_VEL
LIN {X 0,Y 580.73,Z 432.916,A -85,B 0,C 180,E1 -1711.17,E2 -1711.17} C_VEL
LIN {X 0,Y 580.779,Z 420.331,A -85,B 0,C 180,E1 -1711.408,E2 -1711.408} C_VEL
LIN {X 0,Y 580.926,Z 321.798,A -85,B 0,C 180,E1 -1712.632,E2 -1712.632} C_VEL
LIN {X 0,Y 580.318,Z 318.082,A -85,B 0,C 180,E1 -1712.711,E2 -1712.711} C_VEL
LIN {X 0,Y 580.409,Z 303.473,A -85,B 0,C 180,E1 -1715.21,E2 -1715.21} C_VEL
LIN {X 0,Y 580.533,Z 288.36,A -85,B 0,C 180,E1 -1717.827,E2 -1717.827} C_VEL
LIN {X 0,Y 580.26,Z 283.204,A -85,B 0,C 180,E1 -1718.751,E2 -1718.751} C_VEL
LIN {X 0,Y 580.305,Z 283.196,A -85,B 0,C 180,E1 -1721.19,E2 -1721.19} C_VEL
LIN {X 0,Y 580.291,Z 283.199,A -85,B 0,C 180,E1 -1724.327,E2 -1724.327} C_VEL
LIN {X 0,Y 580.233,Z 283.202,A -85,B 0,C 180,E1 -1726.899,E2 -1726.899} C_VEL
LIN {X 0,Y 580.276,Z 283.203,A -85,B 0,C 180,E1 -1729.823,E2 -1729.823} C_VEL
LIN {X 0,Y 580.277,Z 283.198,A -85,B 0,C 180,E1 -1732.802,E2 -1732.802} C_VEL
LIN {X 0,Y 580.246,Z 283.201,A -85,B 0,C 180,E1 -1735.082,E2 -1735.082} C_VEL
LIN {X 0,Y 580.249,Z 283.203,A -85,B 0,C 180,E1 -1737.848,E2 -1737.848} C_VEL
LIN {X 0,Y 580.26,Z 283.205,A -85,B 0,C 180,E1 -1740.69,E2 -1740.69} C_VEL
LIN {X 0,Y 580.272,Z 283.197,A -85,B 0,C 180,E1 -1743.311,E2 -1743.311} C_VEL
LIN {X 0,Y 580.221,Z 283.203,A -85,B 0,C 180,E1 -1745.752,E2 -1745.752} C_VEL
LIN {X 0,Y 580.27,Z 283.2,A -85,B 0,C 180,E1 -1748.147,E2 -1748.147} C_VEL
LIN {X 0,Y 580.265,Z 283.208,A -85,B 0,C 180,E1 -1750.845,E2 -1750.845} C_VEL
LIN {X 0,Y 580.229,Z 283.203,A -85,B 0,C 180,E1 -1753.661,E2 -1753.661} C_VEL
LIN {X 0,Y 580.223,Z 283.208,A -85,B 0,C 180,E1 -1756.614,E2 -1756.614} C_VEL
LIN {X 0,Y 580.269,Z 283.206,A -85,B 0,C 180,E1 -1759.154,E2 -1759.154} C_VEL
LIN {X 0,Y 580.267,Z 283.198,A -85,B 0,C 180,E1 -1761.928,E2 -1761.928} C_VEL
LIN {X 0,Y 580.215,Z 283.205,A -85,B 0,C 180,E1 -1764.45,E2 -1764.45} C_VEL
LIN {X 0,Y 580.231,Z 283.208,A -85,B 0,C 180,E1 -1766.971,E2 -1766.971} C_VEL
LIN {X 0,Y 580.237,Z 283.211,A -85,B 0,C 180,E1 -1769.421,E2 -1769.421} C_VEL
LIN {X 0,Y 580.23,Z 283.203,A -85,B 0,C 180,E1 -1772.152,E2 -1772.152} C_VEL
LIN {X 0,Y 580.227,Z 283.204,A -85,B 0,C 180,E1 -1774.916,E2 -1774.916} C_VEL
LIN {X 0,Y 580.272,Z 283.201,A -85,B 0,C 180,E1 -1777.196,E2 -1777.196} C_VEL
LIN {X 0,Y 580.258,Z 283.202,A -85,B 0,C 180,E1 -1780.176,E2 -1780.176} C_VEL
LIN {X 0,Y 580.219,Z 283.205,A -85,B 0,C 180,E1 -1783.113,E2 -1783.113} C_VEL
LIN {X 0,Y 580.297,Z 283.203,A -85,B 0,C 180,E1 -1785.982,E2 -1785.982} C_VEL
LIN {X 0,Y 580.257,Z 283.199,A -85,B 0,C 180,E1 -1788.826,E2 -1788.826} C_VEL
LIN {X 0,Y 580.284,Z 283.199,A -85,B 0,C 180,E1 -1791.643,E2 -1791.643} C_VEL
LIN {X 0,Y 580.295,Z 283.2,A -85,B 0,C 180,E1 -1794.44,E2 -1794.44} C_VEL
LIN {X 0,Y 580.295,Z 283.194,A -85,B 0,C 180,E1 -1797.223,E2 -1797.223} C_VEL
LIN {X 0,Y 580.324,Z 283.196,A -85,B 0,C 180,E1 -1800,E2 -1800} C_VEL
LIN {X 0,Y 580.323,Z 283.195,A -85,B 0,C 180,E1 -1802.776,E2 -1802.776} C_VEL
LIN {X 0,Y 580.281,Z 283.196,A -85,B 0,C 180,E1 -1805.56,E2 -1805.56} C_VEL
LIN {X 0,Y 580.245,Z 283.2,A -85,B 0,C 180,E1 -1807.656,E2 -1807.656} C_VEL
LIN {X 0,Y 580.261,Z 283.206,A -85,B 0,C 180,E1 -1810.467,E2 -1810.467} C_VEL
LIN {X 0,Y 580.281,Z 283.204,A -85,B 0,C 180,E1 -1812.592,E2 -1812.592} C_VEL
LIN {X 0,Y 580.274,Z 283.198,A -85,B 0,C 180,E1 -1815.453,E2 -1815.453} C_VEL
LIN {X 0,Y 580.252,Z 283.2,A -85,B 0,C 180,E1 -1817.626,E2 -1817.626} C_VEL
LIN {X 0,Y 580.268,Z 283.198,A -85,B 0,C 180,E1 -1819.824,E2 -1819.824} C_VEL
LIN {X 0,Y 580.243,Z 283.2,A -85,B 0,C 180,E1 -1822.054,E2 -1822.054} C_VEL
LIN {X 0,Y 580.274,Z 283.207,A -85,B 0,C 180,E1 -1825.081,E2 -1825.081} C_VEL
LIN {X 0,Y 580.279,Z 283.196,A -85,B 0,C 180,E1 -1828.187,E2 -1828.187} C_VEL
LIN {X 0,Y 580.265,Z 283.199,A -85,B 0,C 180,E1 -1830.693,E2 -1830.693} C_VEL
LIN {X 0,Y 580.294,Z 283.204,A -85,B 0,C 180,E1 -1833.317,E2 -1833.317} C_VEL
LIN {X 0,Y 580.235,Z 283.207,A -85,B 0,C 180,E1 -1835.756,E2 -1835.756} C_VEL
LIN {X 0,Y 580.277,Z 283.198,A -85,B 0,C 180,E1 -1838.147,E2 -1838.147} C_VEL
LIN {X 0,Y 580.287,Z 283.195,A -85,B 0,C 180,E1 -1840.845,E2 -1840.845} C_VEL
LIN {X 0,Y 580.263,Z 283.208,A -85,B 0,C 180,E1 -1843.659,E2 -1843.659} C_VEL
LIN {X 0,Y 580.26,Z 283.199,A -85,B 0,C 180,E1 -1846.611,E2 -1846.611} C_VEL
LIN {X 0,Y 580.289,Z 283.195,A -85,B 0,C 180,E1 -1849.157,E2 -1849.157} C_VEL
LIN {X 0,Y 580.283,Z 283.206,A -85,B 0,C 180,E1 -1851.928,E2 -1851.928} C_VEL
LIN {X 0,Y 580.246,Z 283.205,A -85,B 0,C 180,E1 -1854.453,E2 -1854.453} C_VEL
LIN {X 0,Y 580.285,Z 283.196,A -85,B 0,C 180,E1 -1856.976,E2 -1856.976} C_VEL
LIN {X 0,Y 580.286,Z 283.195,A -85,B 0,C 180,E1 -1859.425,E2 -1859.425} C_VEL
LIN {X 0,Y 580.292,Z 283.203,A -85,B 0,C 180,E1 -1862.143,E2 -1862.143} C_VEL
LIN {X 0,Y 580.289,Z 283.199,A -85,B 0,C 180,E1 -1864.92,E2 -1864.92} C_VEL
LIN {X 0,Y 580.314,Z 283.354,A -85,B 0,C 180,E1 -1867.107,E2 -1867.107} C_VEL
LIN {X 0,Y 580.879,Z 287.767,A -85,B 0,C 180,E1 -1867.785,E2 -1867.785} C_VEL
LIN {X 0,Y 580.7,Z 306.387,A -85,B 0,C 180,E1 -1870.521,E2 -1870.521} C_VEL
LIN {X 0,Y 580.551,Z 325.546,A -85,B 0,C 180,E1 -1873.292,E2 -1873.292} C_VEL
LIN {X 0,Y 580.399,Z 346.64,A -85,B 0,C 180,E1 -1876.298,E2 -1876.298} C_VEL
LIN {X 0,Y 580.416,Z 347.195,A -85,B 0,C 180,E1 -1876.343,E2 -1876.343} C_VEL
LIN {X 0,Y 580.978,Z 352.561,A -85,B 0,C 180,E1 -1876.424,E2 -1876.424} C_VEL
LIN {X 0,Y 580.809,Z 454.979,A -85,B 0,C 180,E1 -1877.709,E2 -1877.709} C_VEL
LIN {X 0,Y 580.733,Z 468.241,A -85,B 0,C 180,E1 -1878.018,E2 -1878.018} C_VEL
LIN {X 0,Y 580.628,Z 481.147,A -85,B 0,C 180,E1 -1878.466,E2 -1878.466} C_VEL
LIN {X 0,Y 580.561,Z 492.64,A -85,B 0,C 180,E1 -1879.009,E2 -1879.009} C_VEL
LIN {X 0,Y 580.437,Z 504.212,A -85,B 0,C 180,E1 -1879.713,E2 -1879.713} C_VEL
LIN {X 0,Y 580.34,Z 514.561,A -85,B 0,C 180,E1 -1880.503,E2 -1880.503} C_VEL
LIN {X 0,Y 580.262,Z 523.062,A -85,B 0,C 180,E1 -1881.293,E2 -1881.293} C_VEL
LIN {X 0,Y 580.221,Z 530.965,A -85,B 0,C 180,E1 -1882.169,E2 -1882.169} C_VEL
LIN {X 0,Y 580.155,Z 538.64,A -85,B 0,C 180,E1 -1883.22,E2 -1883.22} C_VEL
LIN {X 0,Y 580.139,Z 545.683,A -85,B 0,C 180,E1 -1884.439,E2 -1884.439} C_VEL
LIN {X 0,Y 580.108,Z 550.374,A -85,B 0,C 180,E1 -1885.484,E2 -1885.484} C_VEL
LIN {X 0,Y 580.123,Z 553.959,A -85,B 0,C 180,E1 -1886.528,E2 -1886.528} C_VEL
LIN {X 0,Y 580.043,Z 555.81,A -85,B 0,C 180,E1 -1887.223,E2 -1887.223} C_VEL
LIN {X 0,Y 580.038,Z 557.2,A -85,B 0,C 180,E1 -1887.917,E2 -1887.917} C_VEL
LIN {X 0,Y 580.04,Z 558.785,A -85,B 0,C 180,E1 -1889.306,E2 -1889.306} C_VEL
LIN {X 0,Y 580.037,Z 559,A -85,B 0,C 180,E1 -1890.001,E2 -1890.001} C_VEL
LIN {X 0,Y 580.047,Z 558.185,A -85,B 0,C 180,E1 -1891.389,E2 -1891.389} C_VEL
LIN {X 0,Y 580.038,Z 557.199,A -85,B 0,C 180,E1 -1892.084,E2 -1892.084} C_VEL
LIN {X 0,Y 580.043,Z 555.809,A -85,B 0,C 180,E1 -1892.778,E2 -1892.778} C_VEL
LIN {X 0,Y 580.109,Z 552.894,A -85,B 0,C 180,E1 -1893.821,E2 -1893.821} C_VEL
LIN {X 0,Y 580.054,Z 548.947,A -85,B 0,C 180,E1 -1894.866,E2 -1894.866} C_VEL
LIN {X 0,Y 580.14,Z 542.874,A -85,B 0,C 180,E1 -1896.085,E2 -1896.085} C_VEL
LIN {X 0,Y 580.184,Z 536.234,A -85,B 0,C 180,E1 -1897.133,E2 -1897.133} C_VEL
LIN {X 0,Y 580.246,Z 527.987,A -85,B 0,C 180,E1 -1898.182,E2 -1898.182} C_VEL
LIN {X 0,Y 580.333,Z 517.586,A -85,B 0,C 180,E1 -1899.234,E2 -1899.234} C_VEL
LIN {X 0,Y 580.427,Z 507.921,A -85,B 0,C 180,E1 -1900.024,E2 -1900.024} C_VEL
LIN {X 0,Y 580.533,Z 497.32,A -85,B 0,C 180,E1 -1900.728,E2 -1900.728} C_VEL
LIN {X 0,Y 580.646,Z 485.105,A -85,B 0,C 180,E1 -1901.36,E2 -1901.36} C_VEL
LIN {X 0,Y 580.704,Z 473.161,A -85,B 0,C 180,E1 -1901.829,E2 -1901.829} C_VEL
LIN {X 0,Y 580.764,Z 460.503,A -85,B 0,C 180,E1 -1902.182,E2 -1902.182} C_VEL
LIN {X 0,Y 580.829,Z 447.278,A -85,B 0,C 180,E1 -1902.403,E2 -1902.403} C_VEL
LIN {X 0,Y 580.786,Z 349.572,A -85,B 0,C 180,E1 -1903.618,E2 -1903.618} C_VEL
LIN {X 0,Y 580.383,Z 346.79,A -85,B 0,C 180,E1 -1903.681,E2 -1903.681} C_VEL
LIN {X 0,Y 580.552,Z 325.539,A -85,B 0,C 180,E1 -1906.709,E2 -1906.709} C_VEL
LIN {X 0,Y 580.699,Z 306.383,A -85,B 0,C 180,E1 -1909.479,E2 -1909.479} C_VEL
LIN {X 0,Y 580.901,Z 287.759,A -85,B 0,C 180,E1 -1912.215,E2 -1912.215} C_VEL
LIN {X 0,Y 580.279,Z 283.205,A -85,B 0,C 180,E1 -1912.925,E2 -1912.925} C_VEL
LIN {X 0,Y 580.279,Z 283.205,A -85,B 0,C 180,E1 -1915.85,E2 -1915.85} C_VEL
LIN {X 0,Y 580.295,Z 283.199,A -85,B 0,C 180,E1 -1918.186,E2 -1918.186} C_VEL
LIN {X 0,Y 580.278,Z 283.198,A -85,B 0,C 180,E1 -1920.693,E2 -1920.693} C_VEL
LIN {X 0,Y 580.304,Z 283.195,A -85,B 0,C 180,E1 -1923.316,E2 -1923.316} C_VEL
LIN {X 0,Y 580.244,Z 283.208,A -85,B 0,C 180,E1 -1925.756,E2 -1925.756} C_VEL
LIN {X 0,Y 580.287,Z 283.206,A -85,B 0,C 180,E1 -1928.147,E2 -1928.147} C_VEL
LIN {X 0,Y 580.295,Z 283.196,A -85,B 0,C 180,E1 -1930.844,E2 -1930.844} C_VEL
LIN {X 0,Y 580.243,Z 283.202,A -85,B 0,C 180,E1 -1933.661,E2 -1933.661} C_VEL
LIN {X 0,Y 580.267,Z 283.206,A -85,B 0,C 180,E1 -1936.611,E2 -1936.611} C_VEL
LIN {X 0,Y 580.296,Z 283.196,A -85,B 0,C 180,E1 -1939.156,E2 -1939.156} C_VEL
LIN {X 0,Y 580.287,Z 283.195,A -85,B 0,C 180,E1 -1941.928,E2 -1941.928} C_VEL
LIN {X 0,Y 580.249,Z 283.206,A -85,B 0,C 180,E1 -1944.452,E2 -1944.452} C_VEL
LIN {X 0,Y 580.288,Z 283.203,A -85,B 0,C 180,E1 -1946.975,E2 -1946.975} C_VEL
LIN {X 0,Y 580.285,Z 283.198,A -85,B 0,C 180,E1 -1949.424,E2 -1949.424} C_VEL
LIN {X 0,Y 580.288,Z 283.195,A -85,B 0,C 180,E1 -1952.143,E2 -1952.143} C_VEL
LIN {X 0,Y 580.288,Z 283.202,A -85,B 0,C 180,E1 -1954.919,E2 -1954.919} C_VEL
LIN {X 0,Y 580.258,Z 283.199,A -85,B 0,C 180,E1 -1957.947,E2 -1957.947} C_VEL
LIN {X 0,Y 580.3,Z 283.197,A -85,B 0,C 180,E1 -1960.913,E2 -1960.913} C_VEL
LIN {X 0,Y 580.271,Z 283.202,A -85,B 0,C 180,E1 -1963.825,E2 -1963.825} C_VEL
LIN {X 0,Y 580.313,Z 283.195,A -85,B 0,C 180,E1 -1965.983,E2 -1965.983} C_VEL
LIN {X 0,Y 580.306,Z 283.192,A -85,B 0,C 180,E1 -1968.827,E2 -1968.827} C_VEL
LIN {X 0,Y 580.308,Z 283.201,A -85,B 0,C 180,E1 -1971.644,E2 -1971.644} C_VEL
LIN {X 0,Y 580.276,Z 283.205,A -85,B 0,C 180,E1 -1973.742,E2 -1973.742} C_VEL
LIN {X 0,Y 580.27,Z 283.206,A -85,B 0,C 180,E1 -1975.833,E2 -1975.833} C_VEL
LIN {X 0,Y 580.343,Z 283.197,A -85,B 0,C 180,E1 -1977.918,E2 -1977.918} C_VEL
LIN {X 0,Y 580.345,Z 283.189,A -85,B 0,C 180,E1 -1980.694,E2 -1980.694} C_VEL
LIN {X 0,Y 580.323,Z 283.192,A -85,B 0,C 180,E1 -1982.777,E2 -1982.777} C_VEL
LIN {X 0,Y 580.315,Z 283.191,A -85,B 0,C 180,E1 -1985.56,E2 -1985.56} C_VEL
LIN {X 0,Y 580.325,Z 283.201,A -85,B 0,C 180,E1 -1988.356,E2 -1988.356} C_VEL
LIN {X 0,Y 580.302,Z 283.194,A -85,B 0,C 180,E1 -1991.191,E2 -1991.191} C_VEL
LIN {X 0,Y 580.322,Z 283.192,A -85,B 0,C 180,E1 -1994.017,E2 -1994.017} C_VEL
LIN {X 0,Y 580.314,Z 283.199,A -85,B 0,C 180,E1 -1996.914,E2 -1996.914} C_VEL
LIN {X 0,Y 580.284,Z 283.195,A -85,B 0,C 180,E1 -1999.823,E2 -1999.823} C_VEL
LIN {X 0,Y 580.283,Z 283.199,A -85,B 0,C 180,E1 -2001.32,E2 -2001.32} C_VEL
LIN {X 0,Y 579.581,Z 283.285,A -85,B 0,C 180,E1 -2001.9,E2 -2001.9} C_VEL
LIN {X 0,Y 576.699,Z 283.65,A -85,B 0,C 180,E1 -2002.839,E2 -2002.839} C_VEL
LIN {X 0,Y 574.304,Z 283.944,A -85,B 0,C 180,E1 -2003.595,E2 -2003.595} C_VEL
LIN {X 0,Y 573.308,Z 284.065,A -85,B 0,C 180,E1 -2004.179,E2 -2004.179} C_VEL
LIN {X 0,Y 573.243,Z 284.074,A -85,B 0,C 180,E1 -2004.377,E2 -2004.377} C_VEL
LIN {X 0,Y 573.21,Z 284.085,A -85,B 0,C 180,E1 -2006.978,E2 -2006.978} C_VEL
LIN {X 0,Y 573.239,Z 284.079,A -85,B 0,C 180,E1 -2009.487,E2 -2009.487} C_VEL
LIN {X 0,Y 573.252,Z 284.072,A -85,B 0,C 180,E1 -2012.646,E2 -2012.646} C_VEL
LIN {X 0,Y 573.211,Z 284.083,A -85,B 0,C 180,E1 -2015.188,E2 -2015.188} C_VEL
LIN {X 0,Y 573.231,Z 284.08,A -85,B 0,C 180,E1 -2017.808,E2 -2017.808} C_VEL
LIN {X 0,Y 573.248,Z 284.072,A -85,B 0,C 180,E1 -2020.525,E2 -2020.525} C_VEL
LIN {X 0,Y 573.238,Z 284.083,A -85,B 0,C 180,E1 -2023.668,E2 -2023.668} C_VEL
LIN {X 0,Y 573.211,Z 284.078,A -85,B 0,C 180,E1 -2026.638,E2 -2026.638} C_VEL
LIN {X 0,Y 573.249,Z 284.075,A -85,B 0,C 180,E1 -2029.475,E2 -2029.475} C_VEL
LIN {X 0,Y 573.225,Z 284.085,A -85,B 0,C 180,E1 -2032.191,E2 -2032.191} C_VEL
LIN {X 0,Y 573.226,Z 284.076,A -85,B 0,C 180,E1 -2035.231,E2 -2035.231} C_VEL
LIN {X 0,Y 573.242,Z 284.084,A -85,B 0,C 180,E1 -2038.184,E2 -2038.184} C_VEL
LIN {X 0,Y 573.266,Z 284.149,A -85,B 0,C 180,E1 -2039.268,E2 -2039.268} C_VEL
LIN {X 0,Y 573.52,Z 289.319,A -85,B 0,C 180,E1 -2040.194,E2 -2040.194} C_VEL
LIN {X 0,Y 573.404,Z 304.375,A -85,B 0,C 180,E1 -2042.834,E2 -2042.834} C_VEL
LIN {X 0,Y 573.288,Z 318.113,A -85,B 0,C 180,E1 -2045.214,E2 -2045.214} C_VEL
LIN {X 0,Y 574.1,Z 324.087,A -85,B 0,C 180,E1 -2045.322,E2 -2045.322} C_VEL
LIN {X 0,Y 573.874,Z 424.888,A -85,B 0,C 180,E1 -2046.601,E2 -2046.601} C_VEL
LIN {X 0,Y 573.759,Z 438.504,A -85,B 0,C 180,E1 -2046.923,E2 -2046.923} C_VEL
LIN {X 0,Y 573.703,Z 450.612,A -85,B 0,C 180,E1 -2047.349,E2 -2047.349} C_VEL
LIN {X 0,Y 573.528,Z 463.355,A -85,B 0,C 180,E1 -2047.958,E2 -2047.958} C_VEL
LIN {X 0,Y 573.466,Z 474.565,A -85,B 0,C 180,E1 -2048.656,E2 -2048.656} C_VEL
LIN {X 0,Y 573.319,Z 484.88,A -85,B 0,C 180,E1 -2049.457,E2 -2049.457} C_VEL
LIN {X 0,Y 573.254,Z 493.711,A -85,B 0,C 180,E1 -2050.297,E2 -2050.297} C_VEL
LIN {X 0,Y 573.155,Z 501.879,A -85,B 0,C 180,E1 -2051.234,E2 -2051.234} C_VEL
LIN {X 0,Y 573.075,Z 509.585,A -85,B 0,C 180,E1 -2052.33,E2 -2052.33} C_VEL
LIN {X 0,Y 573.041,Z 515.288,A -85,B 0,C 180,E1 -2053.338,E2 -2053.338} C_VEL
LIN {X 0,Y 572.996,Z 519.859,A -85,B 0,C 180,E1 -2054.345,E2 -2054.345} C_VEL
LIN {X 0,Y 572.98,Z 522.55,A -85,B 0,C 180,E1 -2055.073,E2 -2055.073} C_VEL
LIN {X 0,Y 572.996,Z 524.72,A -85,B 0,C 180,E1 -2055.8,E2 -2055.8} C_VEL
LIN {X 0,Y 572.977,Z 526.417,A -85,B 0,C 180,E1 -2056.523,E2 -2056.523} C_VEL
LIN {X 0,Y 572.948,Z 527.685,A -85,B 0,C 180,E1 -2057.244,E2 -2057.244} C_VEL
LIN {X 0,Y 572.948,Z 528.529,A -85,B 0,C 180,E1 -2057.963,E2 -2057.963} C_VEL
LIN {X 0,Y 572.988,Z 528.971,A -85,B 0,C 180,E1 -2058.887,E2 -2058.887} C_VEL
LIN {X 0,Y 572.975,Z 528.539,A -85,B 0,C 180,E1 -2060.112,E2 -2060.112} C_VEL
LIN {X 0,Y 572.928,Z 527.72,A -85,B 0,C 180,E1 -2060.824,E2 -2060.824} C_VEL
LIN {X 0,Y 572.952,Z 526.481,A -85,B 0,C 180,E1 -2061.535,E2 -2061.535} C_VEL
LIN {X 0,Y 572.992,Z 523.84,A -85,B 0,C 180,E1 -2062.6,E2 -2062.6} C_VEL
LIN {X 0,Y 573.012,Z 520.193,A -85,B 0,C 180,E1 -2063.662,E2 -2063.662} C_VEL
LIN {X 0,Y 573.022,Z 515.445,A -85,B 0,C 180,E1 -2064.722,E2 -2064.722} C_VEL
LIN {X 0,Y 573.061,Z 509.461,A -85,B 0,C 180,E1 -2065.78,E2 -2065.78} C_VEL
LIN {X 0,Y 573.148,Z 502.032,A -85,B 0,C 180,E1 -2066.836,E2 -2066.836} C_VEL
LIN {X 0,Y 573.201,Z 494.46,A -85,B 0,C 180,E1 -2067.716,E2 -2067.716} C_VEL
LIN {X 0,Y 573.351,Z 485.306,A -85,B 0,C 180,E1 -2068.595,E2 -2068.595} C_VEL
LIN {X 0,Y 573.401,Z 475.287,A -85,B 0,C 180,E1 -2069.385,E2 -2069.385} C_VEL
LIN {X 0,Y 573.556,Z 464.132,A -85,B 0,C 180,E1 -2070.087,E2 -2070.087} C_VEL
LIN {X 0,Y 573.659,Z 451.63,A -85,B 0,C 180,E1 -2070.701,E2 -2070.701} C_VEL
LIN {X 0,Y 573.739,Z 438.709,A -85,B 0,C 180,E1 -2071.162,E2 -2071.162} C_VEL
LIN {X 0,Y 573.833,Z 425.948,A -85,B 0,C 180,E1 -2071.469,E2 -2071.469} C_VEL
LIN {X 0,Y 574.004,Z 371.711,A -85,B 0,C 180,E1 -2072.17,E2 -2072.17} C_VEL
LIN {X 0,Y 573.944,Z 322.176,A -85,B 0,C 180,E1 -2072.796,E2 -2072.796} C_VEL
LIN {X 0,Y 573.264,Z 318.118,A -85,B 0,C 180,E1 -2072.876,E2 -2072.876} C_VEL
LIN {X 0,Y 573.399,Z 304.271,A -85,B 0,C 180,E1 -2075.274,E2 -2075.274} C_VEL
LIN {X 0,Y 573.548,Z 289.159,A -85,B 0,C 180,E1 -2077.923,E2 -2077.923} C_VEL
LIN {X 0,Y 573.231,Z 284.08,A -85,B 0,C 180,E1 -2078.859,E2 -2078.859} C_VEL
LIN {X 0,Y 573.276,Z 284.073,A -85,B 0,C 180,E1 -2081.311,E2 -2081.311} C_VEL
LIN {X 0,Y 573.267,Z 284.072,A -85,B 0,C 180,E1 -2084.416,E2 -2084.416} C_VEL
LIN {X 0,Y 573.182,Z 284.08,A -85,B 0,C 180,E1 -2087.113,E2 -2087.113} C_VEL
LIN {X 0,Y 573.268,Z 284.07,A -85,B 0,C 180,E1 -2089.329,E2 -2089.329} C_VEL
LIN {X 0,Y 573.217,Z 284.084,A -85,B 0,C 180,E1 -2092.338,E2 -2092.338} C_VEL
LIN {X 0,Y 573.21,Z 284.078,A -85,B 0,C 180,E1 -2094.864,E2 -2094.864} C_VEL
LIN {X 0,Y 573.227,Z 284.076,A -85,B 0,C 180,E1 -2097.767,E2 -2097.767} C_VEL
LIN {X 0,Y 573.223,Z 284.082,A -85,B 0,C 180,E1 -2100.177,E2 -2100.177} C_VEL
LIN {X 0,Y 573.244,Z 284.081,A -85,B 0,C 180,E1 -2102.645,E2 -2102.645} C_VEL
LIN {X 0,Y 573.184,Z 284.082,A -85,B 0,C 180,E1 -2105.188,E2 -2105.188} C_VEL
LIN {X 0,Y 573.21,Z 284.077,A -85,B 0,C 180,E1 -2107.808,E2 -2107.808} C_VEL
LIN {X 0,Y 573.242,Z 284.079,A -85,B 0,C 180,E1 -2110.524,E2 -2110.524} C_VEL
LIN {X 0,Y 573.198,Z 284.078,A -85,B 0,C 180,E1 -2113.664,E2 -2113.664} C_VEL
LIN {X 0,Y 573.19,Z 284.085,A -85,B 0,C 180,E1 -2116.636,E2 -2116.636} C_VEL
LIN {X 0,Y 573.24,Z 284.077,A -85,B 0,C 180,E1 -2119.474,E2 -2119.474} C_VEL
LIN {X 0,Y 573.208,Z 284.077,A -85,B 0,C 180,E1 -2122.19,E2 -2122.19} C_VEL
LIN {X 0,Y 573.215,Z 284.087,A -85,B 0,C 180,E1 -2125.23,E2 -2125.23} C_VEL
LIN {X 0,Y 573.196,Z 284.078,A -85,B 0,C 180,E1 -2128.181,E2 -2128.181} C_VEL
LIN {X 0,Y 573.216,Z 284.076,A -85,B 0,C 180,E1 -2130.631,E2 -2130.631} C_VEL
LIN {X 0,Y 573.181,Z 284.091,A -85,B 0,C 180,E1 -2133.517,E2 -2133.517} C_VEL
LIN {X 0,Y 573.19,Z 284.081,A -85,B 0,C 180,E1 -2136.132,E2 -2136.132} C_VEL
LIN {X 0,Y 573.215,Z 284.076,A -85,B 0,C 180,E1 -2138.716,E2 -2138.716} C_VEL
LIN {X 0,Y 573.18,Z 284.086,A -85,B 0,C 180,E1 -2141.41,E2 -2141.41} C_VEL
LIN {X 0,Y 573.182,Z 284.083,A -85,B 0,C 180,E1 -2144.35,E2 -2144.35} C_VEL
LIN {X 0,Y 573.187,Z 284.081,A -85,B 0,C 180,E1 -2146.528,E2 -2146.528} C_VEL
LIN {X 0,Y 573.23,Z 284.076,A -85,B 0,C 180,E1 -2149.402,E2 -2149.402} C_VEL
LIN {X 0,Y 573.209,Z 284.085,A -85,B 0,C 180,E1 -2152.249,E2 -2152.249} C_VEL
LIN {X 0,Y 573.261,Z 284.07,A -85,B 0,C 180,E1 -2155.077,E2 -2155.077} C_VEL
LIN {X 0,Y 573.284,Z 284.072,A -85,B 0,C 180,E1 -2157.892,E2 -2157.892} C_VEL
LIN {X 0,Y 573.318,Z 284.068,A -85,B 0,C 180,E1 -2160.702,E2 -2160.702} C_VEL
LIN {X 0,Y 573.287,Z 284.071,A -85,B 0,C 180,E1 -2162.811,E2 -2162.811} C_VEL
LIN {X 0,Y 573.251,Z 284.072,A -85,B 0,C 180,E1 -2165.628,E2 -2165.628} C_VEL
LIN {X 0,Y 573.202,Z 284.078,A -85,B 0,C 180,E1 -2167.751,E2 -2167.751} C_VEL
LIN {X 0,Y 573.235,Z 284.083,A -85,B 0,C 180,E1 -2170.597,E2 -2170.597} C_VEL
LIN {X 0,Y 573.203,Z 284.078,A -85,B 0,C 180,E1 -2173.471,E2 -2173.471} C_VEL
LIN {X 0,Y 573.227,Z 284.078,A -85,B 0,C 180,E1 -2176.379,E2 -2176.379} C_VEL
LIN {X 0,Y 573.256,Z 284.075,A -85,B 0,C 180,E1 -2179.33,E2 -2179.33} C_VEL
LIN {X 0,Y 573.211,Z 284.077,A -85,B 0,C 180,E1 -2182.339,E2 -2182.339} C_VEL
LIN {X 0,Y 573.223,Z 284.081,A -85,B 0,C 180,E1 -2185.412,E2 -2185.412} C_VEL
LIN {X 0,Y 573.219,Z 284.077,A -85,B 0,C 180,E1 -2188.566,E2 -2188.566} C_VEL
LIN {X 0,Y 573.213,Z 284.082,A -85,B 0,C 180,E1 -2190.994,E2 -2190.994} C_VEL
LIN {X 0,Y 573.255,Z 284.08,A -85,B 0,C 180,E1 -2193.525,E2 -2193.525} C_VEL
LIN {X 0,Y 573.185,Z 284.082,A -85,B 0,C 180,E1 -2196.054,E2 -2196.054} C_VEL
LIN {X 0,Y 573.229,Z 284.074,A -85,B 0,C 180,E1 -2198.703,E2 -2198.703} C_VEL
LIN {X 0,Y 573.22,Z 284.085,A -85,B 0,C 180,E1 -2201.593,E2 -2201.593} C_VEL
LIN {X 0,Y 573.216,Z 284.078,A -85,B 0,C 180,E1 -2204.335,E2 -2204.335} C_VEL
LIN {X 0,Y 573.227,Z 284.078,A -85,B 0,C 180,E1 -2207.36,E2 -2207.36} C_VEL
LIN {X 0,Y 573.232,Z 284.077,A -85,B 0,C 180,E1 -2210.393,E2 -2210.393} C_VEL
LIN {X 0,Y 573.227,Z 284.075,A -85,B 0,C 180,E1 -2213.077,E2 -2213.077} C_VEL
LIN {X 0,Y 573.26,Z 284.074,A -85,B 0,C 180,E1 -2215.672,E2 -2215.672} C_VEL
LIN {X 0,Y 573.242,Z 284.084,A -85,B 0,C 180,E1 -2218.186,E2 -2218.186} C_VEL
LIN {X 0,Y 573.24,Z 284.078,A -85,B 0,C 180,E1 -2220.634,E2 -2220.634} C_VEL
LIN {X 0,Y 573.219,Z 284.078,A -85,B 0,C 180,E1 -2223.023,E2 -2223.023} C_VEL
LIN {X 0,Y 573.235,Z 284.076,A -85,B 0,C 180,E1 -2225.365,E2 -2225.365} C_VEL
LIN {X 0,Y 573.226,Z 284.118,A -85,B 0,C 180,E1 -2226.949,E2 -2226.949} C_VEL
LIN {X 0,Y 573.952,Z 288.925,A -85,B 0,C 180,E1 -2227.692,E2 -2227.692} C_VEL
LIN {X 0,Y 573.748,Z 308.551,A -85,B 0,C 180,E1 -2230.596,E2 -2230.596} C_VEL
LIN {X 0,Y 573.551,Z 328.092,A -85,B 0,C 180,E1 -2233.452,E2 -2233.452} C_VEL
LIN {X 0,Y 573.422,Z 347.195,A -85,B 0,C 180,E1 -2236.173,E2 -2236.173} C_VEL
